VAR_GLOBAL
	// Interface ID for interface ITcVnCustomContainerOperation_ITcVnContainer
	{attribute 'tc_no_symbol'}
	IID_ITcVnCustomContainerOperation_ITcVnContainer: IID := (Data1 := 16#1324AA81, Data2 := 16#A16E, Data3 := 16#46B2, Data4 := [16#92, 16#D8, 16#11, 16#BE, 16#05, 16#66, 16#C7, 16#7A]);
	// Interface ID for interface ITcVnCustomContainerOperation_ITcVnForwardIterator
	{attribute 'tc_no_symbol'}
	IID_ITcVnCustomContainerOperation_ITcVnForwardIterator: IID := (Data1 := 16#C808A039, Data2 := 16#2D00, Data3 := 16#4B6B, Data4 := [16#89, 16#91, 16#24, 16#B1, 16#F3, 16#3D, 16#98, 16#7A]);
	// Interface ID for interface ITcVnCustomElementCondition_ITcVnContainer
	{attribute 'tc_no_symbol'}
	IID_ITcVnCustomElementCondition_ITcVnContainer: IID := (Data1 := 16#2529A58B, Data2 := 16#9E91, Data3 := 16#49A1, Data4 := [16#AD, 16#8A, 16#95, 16#06, 16#B8, 16#87, 16#F0, 16#65]);
	// Interface ID for interface ITcVnCustomElementCondition_ITcVnForwardIterator
	{attribute 'tc_no_symbol'}
	IID_ITcVnCustomElementCondition_ITcVnForwardIterator: IID := (Data1 := 16#7CF2DF09, Data2 := 16#9C9A, Data3 := 16#4433, Data4 := [16#98, 16#DD, 16#BF, 16#28, 16#40, 16#7D, 16#A3, 16#D4]);
	// Interface ID for interface ITcVnColorModel
	{attribute 'tc_no_symbol'}
	IID_ITcVnColorModel: IID := (Data1 := 16#0D1C5AC3, Data2 := 16#B759, Data3 := 16#4DFF, Data4 := [16#86, 16#24, 16#65, 16#78, 16#26, 16#E9, 16#F5, 16#8E]);
END_VAR

// Version/Global_Version
{attribute 'TcGenerated'}
// This function has been automatically generated from the project information.
VAR_GLOBAL CONSTANT
	{attribute 'const_non_replaced'}
	{attribute 'linkalways'}
	stLibVersion_Tc3_Vision : ST_LibVersion := (iMajor := 3, iMinor := 1, iBuild := 1, iRevision := 12, sVersion := '3.1.1.12');
	{attribute 'const_non_replaced'}
	{attribute 'linkalways'}
	sLibraryId_Tc3_Vision : String := 'Beckhoff Automation GmbH|Tc3_Vision|3.1.1.12';
END_VAR

// Global Variables/Global_Variables

	VAR_GLOBAL
		VISION_ADS_TIMEOUT	:	TIME := TIME#5s;	(* Default ADS timeout. *)
	END_VAR

// Function Blocks/Image Acquisition/FB_VN_GevCameraControl

	{attribute 'c++_compatible'}
	{attribute 'external_name' := 'FB_VN_GevCameraControl_GUID_F17A7C37_E616_4417_46AF_6CAA272D4BB4'}
	{attribute 'TcIecLibraryType'}
	(* This FB provides the basic functionality to control a GigE Vision camera and access its calibration data. *)
	FUNCTION_BLOCK FB_VN_GevCameraControl
	VAR
		(* Internal reference to the corresponding TcVnGevImageProvider TcCOM module ID, which needs to be set via TC init symbol. *)
		{attribute 'TcInitSymbol'}
		{attribute 'TcCategoryOID' := 'TcVnGevImageProvider'}
		 {attribute 'GUID' := '18071995-0000-0000-0000-00000000000F'}
		oidITcVnGevImageProvider : OTCID;
		 {attribute 'hide'}
		_reserved1 : UINT_0_32;
		(* Internal stuff *)
		{attribute 'hide'}
		 {attribute 'GUID' := '18071995-0000-0000-0000-000000000018'}
		pInternal : PVOID;
	END_VAR


	(* Delete all images contained in the TcVnGevImageProvider TcCOM module receive queue and reset the corresponding omitted images counter. *)
	METHOD ClearImageQueue : HRESULT
END_METHOD


	(* Close the control channel to the camera. *)
	METHOD CloseCamera : HRESULT
END_METHOD


	(* Internal method *)
	{attribute 'hide'}
	METHOD FB_exit : BOOL
	VAR_INPUT
		(*  if TRUE, the exit method is called for exiting an instance that is copied afterwards (online change). *)
		bInCopyCode : BOOL;
	END_VAR
END_METHOD


	(* Internal method *)
	{attribute 'hide'}
	METHOD FB_init : BOOL
	VAR_INPUT
		(*  if TRUE, the retain variables are initialized (warm start / cold start) *)
		bInitRetains : BOOL;
		(*  if TRUE, the instance afterwards gets moved into the copy code (online change) *)
		bInCopyCode : BOOL;
	END_VAR
END_METHOD


	(* Gets the reference calibration pattern points from the TcVnGevImageProvider TcCOM module (Can be set from the calibration assistant) *)
	METHOD GetCalibPatternRef : HRESULT
	VAR_INPUT
		(* Returns the reference calibration pattern points (ContainerType_Vector_TcVnPoint3_REAL) *)
 {attribute 'GUID' := 'BC72B333-E095-465B-9693-7979773CA3B8'}
				ipCalibPatternRef : REFERENCE TO ITcVnContainer;
	END_VAR
END_METHOD


	(* Gets the camera matrix from the TcVnGevImageProvider TcCOM module (requires intrinsic calibration parameters, e.g. set by the calibration assistant) *)
	METHOD GetCameraMatrix : HRESULT
	VAR_INPUT
		(* Returns the camera matrix *)
 {attribute 'GUID' := '91A420A3-4727-4481-B3BB-170528E5BC7C'}
		 {attribute 'Namespace' := 'VN'}
				aCameraMatrix : REFERENCE TO TcVnMatrix3x3_LREAL;
	END_VAR
END_METHOD


	(* Gets the current available image (first in receive queue). *)
	METHOD GetCurrentImage : HRESULT
	VAR_INPUT
		(* Returns the image *)
 {attribute 'GUID' := '70D42C6D-6F4E-4719-8B29-2883D5D59B1C'}
				ipImage : REFERENCE TO ITcVnImage;
	END_VAR
END_METHOD


	(* Gets the current available image (first in receive queue) with undistortion applied (requires intrinsic calibration parameters in the TcVnGevImageProvider TcCOM module, e.g. set by the calibration assistant) *)
	METHOD GetCurrentImageUndistorted : HRESULT
	VAR_INPUT
		(* Returns the undistorted image *)
 {attribute 'GUID' := '70D42C6D-6F4E-4719-8B29-2883D5D59B1C'}
				ipImage : REFERENCE TO ITcVnImage;
	END_VAR
END_METHOD


	(* Gets the current available image (first in receive queue) and its corresponding GVSP info. *)
	METHOD GetCurrentImageWithGvspInfo : HRESULT
	VAR_INPUT
		(* Returns the image *)
 {attribute 'GUID' := '70D42C6D-6F4E-4719-8B29-2883D5D59B1C'}
				ipImage : REFERENCE TO ITcVnImage;
		(* Returns the GVSP info *)
 {attribute 'GUID' := '63FC7E33-91CD-44CD-9015-0BD1DC25722C'}
				stGvspInfo : REFERENCE TO GVSP_IMAGE_INFO;
	END_VAR
END_METHOD


	(* Gets the current available image (first in receive queue) with its corresponding GVSP info and undistortion applied (requires intrinsic calibration parameters in the TcVnGevImageProvider TcCOM module, e.g. set by the calibration assistant) *)
	METHOD GetCurrentImageWithGvspInfoUndistorted : HRESULT
	VAR_INPUT
		(* Returns the undistorted image *)
 {attribute 'GUID' := '70D42C6D-6F4E-4719-8B29-2883D5D59B1C'}
				ipImage : REFERENCE TO ITcVnImage;
		(* Returns the GVSP info *)
 {attribute 'GUID' := '63FC7E33-91CD-44CD-9015-0BD1DC25722C'}
				stGvspInfo : REFERENCE TO GVSP_IMAGE_INFO;
	END_VAR
END_METHOD


	(* Gets the distortion coefficients from the TcVnGevImageProvider TcCOM module (requires intrinsic calibration parameters, e.g. set by the calibration assistant) *)
	METHOD GetDistortionCoefficients : HRESULT
	VAR_INPUT
		(* Returns the distortion coefficients [k1, k2, p1, p2, k3, k4, k5, k6] *)
 {attribute 'GUID' := 'DD112102-C23A-4B37-A43A-A96400B57010'}
		 {attribute 'Namespace' := 'VN'}
				aDistortionCoefficients : REFERENCE TO TcVnArray8_LREAL;
	END_VAR
END_METHOD


	(* Gets the last received image from the queue. *)
	METHOD GetLastImageFromQueue : HRESULT
	VAR_INPUT
		(* Returns the image *)
 {attribute 'GUID' := '70D42C6D-6F4E-4719-8B29-2883D5D59B1C'}
				ipImage : REFERENCE TO ITcVnImage;
	END_VAR
END_METHOD


	(* Gets the number of omitted images since the last call of ClearImageQueue(). If the image receive queue in the TcVnGevImageProvider TcCOM module is full and a new image arrives, the first one in the queue will be deleted and the omitted counter is increased. *)
	METHOD GetOmittedImagesNum : HRESULT
	VAR_INPUT
		(* Returns the number of omitted images *)
		nOmitted : REFERENCE TO ULINT;
	END_VAR
END_METHOD


	(* Gets the rotation matrix from the TcVnGevImageProvider TcCOM module (requires extrinsic calibration parameters, e.g. set by the calibration assistant) *)
	METHOD GetRotationMatrix : HRESULT
	VAR_INPUT
		(* Returns the rotation matrix *)
 {attribute 'GUID' := '91A420A3-4727-4481-B3BB-170528E5BC7C'}
		 {attribute 'Namespace' := 'VN'}
				aRotationMatrix : REFERENCE TO TcVnMatrix3x3_LREAL;
	END_VAR
END_METHOD


	(* Gets the current state of the internal camera control state machine. *)
	METHOD GetState : ETcVnCameraState
END_METHOD


	(* Gets the translation vector from the TcVnGevImageProvider TcCOM module (requires extrinsic calibration parameters, e.g. set by the calibration assistant) *)
	METHOD GetTranslationVector : HRESULT
	VAR_INPUT
		(* Returns the translation vector *)
 {attribute 'GUID' := 'B9A67DEB-A7D1-4F25-95A3-4A82FA5C1E28'}
		 {attribute 'Namespace' := 'VN'}
				aTranslationVector : REFERENCE TO TcVnVector3_LREAL;
	END_VAR
END_METHOD


	(* Initialize the camera to the intended state (includes sending the 'InitCameraCommands' defined in the GevImageAcquisition TcCOM module to the camera). *)
	METHOD InitializeCamera : HRESULT
END_METHOD


	(* Open a control channel to the camera. *)
	METHOD OpenCamera : HRESULT
END_METHOD


	(* Reset the camera controller to initial state (might require multiple calls depending on current state, until S_OK is returned) *)
	METHOD Reset : HRESULT
END_METHOD


	(* Reset the camera features to initial state (sends the 'InitCameraCommands' defined in the GevImageAcquisition TcCOM module to the camera). *)
	METHOD ResetCameraFeatures : HRESULT
END_METHOD


	(* Sets the camera matrix to the TcVnGevImageProvider TcCOM module *)
	METHOD SetCameraMatrix : HRESULT
	VAR_INPUT
		(* The camera matrix to be copied to the TcCOM module *)
 {attribute 'GUID' := '91A420A3-4727-4481-B3BB-170528E5BC7C'}
		 {attribute 'Namespace' := 'VN'}
				aCameraMatrix : REFERENCE TO TcVnMatrix3x3_LREAL;
	END_VAR
END_METHOD


	(* Sets the distortion coefficients to the TcVnGevImageProvider TcCOM module *)
	METHOD SetDistortionCoefficients : HRESULT
	VAR_INPUT
		(* The distortion coefficients to be copied to the TcCOM module *)
 {attribute 'GUID' := 'DD112102-C23A-4B37-A43A-A96400B57010'}
		 {attribute 'Namespace' := 'VN'}
				aDistortionCoefficients : REFERENCE TO TcVnArray8_LREAL;
	END_VAR
END_METHOD


	(* Sets the rotation matrix to the TcVnGevImageProvider TcCOM module *)
	METHOD SetRotationMatrix : HRESULT
	VAR_INPUT
		(* The rotation matrix to be copied to the TcCOM module *)
 {attribute 'GUID' := '91A420A3-4727-4481-B3BB-170528E5BC7C'}
		 {attribute 'Namespace' := 'VN'}
				aRotationMatrix : REFERENCE TO TcVnMatrix3x3_LREAL;
	END_VAR
END_METHOD


	(* Sets the translation vector to the TcVnGevImageProvider TcCOM module *)
	METHOD SetTranslationVector : HRESULT
	VAR_INPUT
		(* The translation vector to be copied to the TcCOM module *)
 {attribute 'GUID' := 'B9A67DEB-A7D1-4F25-95A3-4A82FA5C1E28'}
		 {attribute 'Namespace' := 'VN'}
				aTranslationVector : REFERENCE TO TcVnVector3_LREAL;
	END_VAR
END_METHOD


	(* Send the 'StartAcquisitionCommands' defined in the TcVnGevImageProvider TcCOM module to the camera. *)
	METHOD StartAcquisition : HRESULT
END_METHOD


	(* Send the 'StopAcquisitionCommands' defined in the TcVnGevImageProvider TcCOM module to the camera. *)
	METHOD StopAcquisition : HRESULT
END_METHOD


	(* Send the 'SoftwareTriggerCommands' defined in the TcVnGevImageProvider TcCOM module to the camera. *)
	METHOD TriggerImage : HRESULT
END_METHOD

END_FUNCTION_BLOCK

// Function Blocks/Image Acquisition/FB_VN_FileSourceControl

	{attribute 'c++_compatible'}
	{attribute 'external_name' := 'FB_VN_FileSourceControl_GUID_0F8A3DBC_2DD8_48DE_55D7_61CBFB8E01C0'}
	{attribute 'TcIecLibraryType'}
	(* This FB provides access to the images send by a File SOurce instance. *)
	FUNCTION_BLOCK FB_VN_FileSourceControl
	VAR
		(* Internal reference to the corresponding TcVnFileImageProvider TcCOM module ID, which needs to be set via TC init symbol. *)
		{attribute 'TcInitSymbol'}
		{attribute 'TcCategoryOID' := 'TcVnFileImageProvider'}
		 {attribute 'GUID' := '18071995-0000-0000-0000-00000000000F'}
		oidITcVnFileImageProvider : OTCID;
		 {attribute 'hide'}
		_reserved1 : UINT_0_32;
		(* Internal reference to private data. *)
		{attribute 'hide'}
		 {attribute 'GUID' := '18071995-0000-0000-0000-000000000018'}
		pPriv : PVOID;
	END_VAR


	(* Internal method *)
	{attribute 'hide'}
	METHOD FB_exit : BOOL
	VAR_INPUT
		(* If TRUE, the exit method is called for exiting an instance that is copied afterwards (online change). *)
		bInCopyCode : BOOL;
	END_VAR
END_METHOD


	(* Internal method *)
	{attribute 'hide'}
	METHOD FB_init : BOOL
	VAR_INPUT
		(* If TRUE, the retain variables are initialized (warm start / cold start) *)
		bInitRetains : BOOL;
		(* If TRUE, the exit method is called for exiting an instance that is copied afterwards (online change). *)
		bInCopyCode : BOOL;
	END_VAR
END_METHOD


	(* Gets the current available image (if any). *)
	METHOD GetCurrentImage : HRESULT
	VAR_INPUT
		(* Returns the image *)
 {attribute 'GUID' := '70D42C6D-6F4E-4719-8B29-2883D5D59B1C'}
				ipImage : REFERENCE TO ITcVnImage;
	END_VAR
END_METHOD


	(* Gets the current available image (if any) and the corresponding file name. *)
	METHOD GetCurrentImageAndFileName : HRESULT
	VAR_INPUT
		(* Returns the image *)
 {attribute 'GUID' := '70D42C6D-6F4E-4719-8B29-2883D5D59B1C'}
				ipImage : REFERENCE TO ITcVnImage;
	END_VAR
	VAR_IN_OUT CONSTANT
		(* Returns the file name *)
 {attribute 'GUID' := '18071995-0000-0000-0000-00000000001A'}
				sFileName : STRING;
	END_VAR
	VAR_INPUT
		(* Define the maximum allowed length for the file name *)
		nMaxLen : UINT;
	END_VAR
END_METHOD


	(* Activates the File Source. If not in trigger mode, it will start sending images. *)
	METHOD StartAcquisition : HRESULT
END_METHOD


	(* Deactivates the File Source. It will stop sending images. *)
	METHOD StopAcquisition : HRESULT
END_METHOD


	(* Reset the controller to initial state (might require multiple calls depending on current state, until S_OK is returned) *)
	METHOD Reset : HRESULT
END_METHOD


	(* Gets the current state of the internal camera control state machine. *)
	METHOD GetState : ETcVnCameraState
END_METHOD


	(* If in trigger mode, this function triggers the next image in the list. *)
	METHOD TriggerImage : HRESULT
END_METHOD


	(* If in trigger mode, this function triggers a specific image in the list. *)
	METHOD TriggerImageExp : HRESULT
	VAR_INPUT
		(* Amount of images to skip, relative to current *)
		nSkipImages : DINT;
	END_VAR
END_METHOD


	(* If in trigger mode, this function triggers a specific image in the list by name. *)
	METHOD TriggerImageByName : HRESULT
	VAR_IN_OUT CONSTANT
		(* Name of the image to trigger *)
 {attribute 'GUID' := '18071995-0000-0000-0000-00000000001A'}
				sImageName : STRING;
	END_VAR
END_METHOD

END_FUNCTION_BLOCK

// Function Blocks/Image Acquisition/FB_VN_SimpleCameraControl

	{attribute 'c++_compatible'}
	{attribute 'external_name' := 'FB_VN_SimpleCameraControl_GUID_85A4A3A7_7C55_424E_46D9_2337A2CE214C'}
	{attribute 'TcIecLibraryType'}
	(* This FB provides the basic functionality to control a camera or a FileSource. *)
	FUNCTION_BLOCK FB_VN_SimpleCameraControl
	VAR
		(* Internal reference to the corresponding TcVnImageProvider TcCOM module ID, which needs to be set via TC init symbol. *)
		{attribute 'TcInitSymbol'}
		{attribute 'TcCategoryOID' := 'TcVnImageProvider'}
		 {attribute 'GUID' := '18071995-0000-0000-0000-00000000000F'}
		oidITcVnImageProvider : OTCID;
		 {attribute 'hide'}
		_reserved1 : UINT_0_32;
		(* Internal stuff *)
		{attribute 'hide'}
		 {attribute 'GUID' := '18071995-0000-0000-0000-000000000018'}
		pInternal : PVOID;
	END_VAR


	(* Internal method *)
	{attribute 'hide'}
	METHOD FB_exit : BOOL
	VAR_INPUT
		(*  if TRUE, the exit method is called for exiting an instance that is copied afterwards (online change). *)
		bInCopyCode : BOOL;
	END_VAR
END_METHOD


	(* Internal method *)
	{attribute 'hide'}
	METHOD FB_init : BOOL
	VAR_INPUT
		(*  if TRUE, the retain variables are initialized (warm start / cold start) *)
		bInitRetains : BOOL;
		(*  if TRUE, the instance afterwards gets moved into the copy code (online change) *)
		bInCopyCode : BOOL;
	END_VAR
END_METHOD


	(* Get the current available image (if any). *)
	METHOD GetCurrentImage : HRESULT
	VAR_INPUT
		(* Returns the image *)
 {attribute 'GUID' := '70D42C6D-6F4E-4719-8B29-2883D5D59B1C'}
				ipImage : REFERENCE TO ITcVnImage;
	END_VAR
END_METHOD


	(* Get the current state of the internal camera control state machine. *)
	METHOD GetState : ETcVnCameraState
END_METHOD


	(* Reset the camera to initial state (might require multiple calls depending on current state, until S_OK is returned) *)
	METHOD Reset : HRESULT
END_METHOD


	(* Start the image acquisition. *)
	METHOD StartAcquisition : HRESULT
END_METHOD


	(* Stop the image acquisition. *)
	METHOD StopAcquisition : HRESULT
END_METHOD


	(* Trigger the next image. *)
	METHOD TriggerImage : HRESULT
END_METHOD

END_FUNCTION_BLOCK

// Function Blocks/File Access/FB_VN_ReadCalibrationPattern

	{attribute 'c++_compatible'}
	{attribute 'external_name' := 'FB_VN_ReadCalibrationPattern_GUID_B3A02584_AB5A_4ACE_53F2_D2DD5DC64051'}
	{attribute 'TcIecLibraryType'}
	(* This FB reads calibration pattern reference points from an xml file on the targte pc. *)
	FUNCTION_BLOCK FB_VN_ReadCalibrationPattern
	VAR_IN_OUT CONSTANT
		(* Full path of the file or relative path to the default directory on the target pc (%TWINCAT3DIR%\\CustomConfig\\Vision\\CalibrationPattern) *)
		 {attribute 'GUID' := '18071995-0000-0000-0000-00000000001A'}
		sFilePath : STRING;
	END_VAR
	VAR_INPUT
		(* Returns a container with the pattern points (ContainerType_Vector_TcVnPoint3_REAL) *)
		 {attribute 'GUID' := 'BC72B333-E095-465B-9693-7979773CA3B8'}
		ipDestContainer : REFERENCE TO ITcVnContainer;
		(* Reading the file is triggered by a rising edge at this input. *)
		bRead : BOOL;
	END_VAR
	VAR
		 {attribute 'hide'}
		_reserved1 : ARRAY [1..3] OF USINT;
	END_VAR
	VAR_INPUT
		(* Indicates the time before the function is cancelled. *)
		nTimeout : TIME := VISION_ADS_TIMEOUT;
	END_VAR
	VAR_OUTPUT
		(* This output remains TRUE until the function block has executed a command, but at the longest for the duration supplied to the 'nTimeout' input. While bBusy = TRUE, no new command will be accepted at the inputs. *)
		bBusy : BOOL;
		(* This output is switched to TRUE as soon as an error occurs during the execution of a command. The command-specific error code is contained in ‘nErrorId’. If the function block has a timeout error, 'bError' is TRUE and 'nErrorId' is 1861 (hexadecimal 0x745). Is reset to FALSE by the execution of a command at the inputs. *)
		bError : BOOL;
	END_VAR
	VAR
		 {attribute 'hide'}
		_reserved2 : UINT;
	END_VAR
	VAR_OUTPUT
		(* Contains the ADS error code or the command-specific error code of the last executed command. Is reset to 0 by the execution of a command at the inputs. *)
		nErrorId : UDINT;
	END_VAR
	VAR
		(* Internal parameter *)
		{attribute 'hide'}
		nAdsInvStamp : UINT;
		(* Internal parameter *)
		{attribute 'hide'}
		nAdsInvCnt : BYTE;
		(* Internal parameter *)
		{attribute 'hide'}
		ePendingRequest : BYTE;
		(* Internal parameter *)
		{attribute 'hide'}
		nTimeElapsed : TIME;
		(* Internal parameter *)
		{attribute 'hide'}
		bLastRead : BOOL;
		 {attribute 'hide'}
		_reserved3 : UINT_24_56;
		(* Internal parameter *)
		{attribute 'hide'}
		 {attribute 'GUID' := '18071995-0000-0000-0000-000000000018'}
		pBuffer : PVOID;
	END_VAR


	(* Internal method *)
	{attribute 'hide'}
	METHOD FB_exit : BOOL
	VAR_INPUT
		(*  if TRUE, the exit method is called for exiting an instance that is copied afterwards (online change). *)
		bInCopyCode : BOOL;
	END_VAR
END_METHOD


	(* Internal method *)
	{attribute 'hide'}
	METHOD FB_init : BOOL
	VAR_INPUT
		(*  if TRUE, the retain variables are initialized (warm start / cold start) *)
		bInitRetains : BOOL;
		(*  if TRUE, the instance afterwards gets moved into the copy code (online change) *)
		bInCopyCode : BOOL;
	END_VAR
END_METHOD

END_FUNCTION_BLOCK

// Function Blocks/File Access/FB_VN_ReadContainer

	{attribute 'c++_compatible'}
	{attribute 'external_name' := 'FB_VN_ReadContainer_GUID_4970374B_76DF_4A68_6AE7_EC922972F9F2'}
	{attribute 'TcIecLibraryType'}
	(* This FB reads a container from an xml file on the target pc. *)
	FUNCTION_BLOCK FB_VN_ReadContainer
	VAR_IN_OUT CONSTANT
		(* Full path of the file or relative path to the default directory on the target pc *)
		 {attribute 'GUID' := '18071995-0000-0000-0000-00000000001A'}
		sFilePath : STRING;
	END_VAR
	VAR_INPUT
		(* Returns a container with the loaded content *)
		 {attribute 'GUID' := 'BC72B333-E095-465B-9693-7979773CA3B8'}
		ipDestContainer : REFERENCE TO ITcVnContainer;
		(* The type id of the container to return. If this parameter is not set, a suitable container type will be determined automatically. *)
		 {attribute 'GUID' := '18071995-0000-0000-0000-000000000021'}
		nDestTypeGuid : GUID;
		(* Reading the file is triggered by a rising edge at this input. *)
		bRead : BOOL;
	END_VAR
	VAR
		 {attribute 'hide'}
		_reserved1 : ARRAY [1..3] OF USINT;
	END_VAR
	VAR_INPUT
		(* Indicates the time before the function is cancelled. *)
		nTimeout : TIME := VISION_ADS_TIMEOUT;
	END_VAR
	VAR_OUTPUT
		(* This output remains TRUE until the function block has executed a command, but at the longest for the duration supplied to the 'nTimeout' input. While bBusy = TRUE, no new command will be accepted at the inputs. *)
		bBusy : BOOL;
		(* This output is switched to TRUE as soon as an error occurs during the execution of a command. The command-specific error code is contained in ‘nErrorId’. If the function block has a timeout error, 'bError' is TRUE and 'nErrorId' is 1861 (hexadecimal 0x745). Is reset to FALSE by the execution of a command at the inputs. *)
		bError : BOOL;
	END_VAR
	VAR
		 {attribute 'hide'}
		_reserved2 : UINT;
	END_VAR
	VAR_OUTPUT
		(* Contains the ADS error code or the command-specific error code of the last executed command. Is reset to 0 by the execution of a command at the inputs. *)
		nErrorId : UDINT;
	END_VAR
	VAR
		(* Internal parameter *)
		{attribute 'hide'}
		nAdsInvStamp : UINT;
		(* Internal parameter *)
		{attribute 'hide'}
		nAdsInvCnt : BYTE;
		(* Internal parameter *)
		{attribute 'hide'}
		ePendingRequest : BYTE;
		(* Internal parameter *)
		{attribute 'hide'}
		nTimeElapsed : TIME;
		(* Internal parameter *)
		{attribute 'hide'}
		bLastRead : BOOL;
		 {attribute 'hide'}
		_reserved3 : UINT_24_56;
		(* Internal parameter *)
		{attribute 'hide'}
		 {attribute 'GUID' := '18071995-0000-0000-0000-000000000018'}
		pBuffer : PVOID;
	END_VAR


	(* Internal method *)
	{attribute 'hide'}
	METHOD FB_exit : BOOL
	VAR_INPUT
		(*  if TRUE, the exit method is called for exiting an instance that is copied afterwards (online change). *)
		bInCopyCode : BOOL;
	END_VAR
END_METHOD


	(* Internal method *)
	{attribute 'hide'}
	METHOD FB_init : BOOL
	VAR_INPUT
		(*  if TRUE, the retain variables are initialized (warm start / cold start) *)
		bInitRetains : BOOL;
		(*  if TRUE, the instance afterwards gets moved into the copy code (online change) *)
		bInCopyCode : BOOL;
	END_VAR
END_METHOD

END_FUNCTION_BLOCK

// Function Blocks/File Access/FB_VN_ReadImage

	{attribute 'c++_compatible'}
	{attribute 'external_name' := 'FB_VN_ReadImage_GUID_DC225DEA_0B37_4A85_7737_55D65C996AC9'}
	{attribute 'TcIecLibraryType'}
	(* This FB reads an image from a file on the target pc. *)
	FUNCTION_BLOCK FB_VN_ReadImage
	VAR_IN_OUT CONSTANT
		(* Full path of the file or relative path to the default image directory on the target pc *)
		 {attribute 'GUID' := '18071995-0000-0000-0000-00000000001A'}
		sFilePath : STRING;
	END_VAR
	VAR_INPUT
		(* Returns an image with the loaded content *)
		 {attribute 'GUID' := '70D42C6D-6F4E-4719-8B29-2883D5D59B1C'}
		ipDestImage : REFERENCE TO ITcVnImage;
		(* Reading the file is triggered by a rising edge at this input. *)
		bRead : BOOL;
	END_VAR
	VAR
		 {attribute 'hide'}
		_reserved1 : ARRAY [1..3] OF USINT;
	END_VAR
	VAR_INPUT
		(* Indicates the time before the function is cancelled. *)
		nTimeout : TIME := VISION_ADS_TIMEOUT;
	END_VAR
	VAR_OUTPUT
		(* This output remains TRUE until the function block has executed a command, but at the longest for the duration supplied to the 'nTimeout' input. While bBusy = TRUE, no new command will be accepted at the inputs. *)
		bBusy : BOOL;
		(* This output is switched to TRUE as soon as an error occurs during the execution of a command. The command-specific error code is contained in ‘nErrorId’. If the function block has a timeout error, 'bError' is TRUE and 'nErrorId' is 1861 (hexadecimal 0x745). Is reset to FALSE by the execution of a command at the inputs. *)
		bError : BOOL;
	END_VAR
	VAR
		 {attribute 'hide'}
		_reserved2 : UINT;
	END_VAR
	VAR_OUTPUT
		(* Contains the ADS error code or the command-specific error code of the last executed command. Is reset to 0 by the execution of a command at the inputs. *)
		nErrorId : UDINT;
	END_VAR
	VAR
		(* Internal parameter *)
		{attribute 'hide'}
		nAdsInvStamp : UINT;
		(* Internal parameter *)
		{attribute 'hide'}
		nAdsInvCnt : BYTE;
		(* Internal parameter *)
		{attribute 'hide'}
		ePendingRequest : BYTE;
		(* Internal parameter *)
		{attribute 'hide'}
		nTimeElapsed : TIME;
		(* Internal parameter *)
		{attribute 'hide'}
		bLastRead : BOOL;
		 {attribute 'hide'}
		_reserved3 : UINT_24_56;
		(* Internal parameter *)
		{attribute 'hide'}
		 {attribute 'GUID' := '18071995-0000-0000-0000-000000000018'}
		pBuffer : PVOID;
	END_VAR


	(* Internal method *)
	{attribute 'hide'}
	METHOD FB_exit : BOOL
	VAR_INPUT
		(*  if TRUE, the exit method is called for exiting an instance that is copied afterwards (online change). *)
		bInCopyCode : BOOL;
	END_VAR
END_METHOD


	(* Internal method *)
	{attribute 'hide'}
	METHOD FB_init : BOOL
	VAR_INPUT
		(*  if TRUE, the retain variables are initialized (warm start / cold start) *)
		bInitRetains : BOOL;
		(*  if TRUE, the instance afterwards gets moved into the copy code (online change) *)
		bInCopyCode : BOOL;
	END_VAR
END_METHOD

END_FUNCTION_BLOCK

// Function Blocks/File Access/FB_VN_WriteContainer

	{attribute 'c++_compatible'}
	{attribute 'external_name' := 'FB_VN_WriteContainer_GUID_7951D962_7694_4A6A_69EC_EB8831476B4E'}
	{attribute 'TcIecLibraryType'}
	(* This FB writes a container as an xml file to the hard drive. *)
	FUNCTION_BLOCK FB_VN_WriteContainer
	VAR_INPUT
		(* The container to write *)
		 {attribute 'GUID' := 'BC72B333-E095-465B-9693-7979773CA3B8'}
		ipContainer : ITcVnContainer;
	END_VAR
	VAR_IN_OUT CONSTANT
		(* Full path of the file or relative path to the default directory on the target pc *)
		 {attribute 'GUID' := '18071995-0000-0000-0000-00000000001A'}
		sFilePath : STRING;
	END_VAR
	VAR_INPUT
		(* Container export format (default is human readable xml) *)
		 {attribute 'GUID' := 'F8305D79-70A3-4F93-A939-2FF3B8D6AF74'}
		 {attribute 'Namespace' := 'Tc3_Vision'}
		eExportFormat : ETcVnContainerExportFormat := TCVN_CEF_XML;
		(* Writing the container is triggered by a rising edge at this input. *)
		bWrite : BOOL;
	END_VAR
	VAR
		 {attribute 'hide'}
		_reserved1 : USINT;
	END_VAR
	VAR_INPUT
		(* Indicates the time before the function is cancelled. *)
		nTimeout : TIME := VISION_ADS_TIMEOUT;
	END_VAR
	VAR_OUTPUT
		(* This output remains TRUE until the function block has executed a command, but at the longest for the duration supplied to the 'nTimeout' input. While bBusy = TRUE, no new command will be accepted at the inputs. *)
		bBusy : BOOL;
		(* This output is switched to TRUE as soon as an error occurs during the execution of a command. The command-specific error code is contained in ‘nErrorId’. If the function block has a timeout error, 'bError' is TRUE and 'nErrorId' is 1861 (hexadecimal 0x745). Is reset to FALSE by the execution of a command at the inputs. *)
		bError : BOOL;
	END_VAR
	VAR
		 {attribute 'hide'}
		_reserved2 : UINT;
	END_VAR
	VAR_OUTPUT
		(* Contains the ADS error code or the command-specific error code of the last executed command. Is reset to 0 by the execution of a command at the inputs. *)
		nErrorId : UDINT;
	END_VAR
	VAR
		(* Internal parameter *)
		{attribute 'hide'}
		nAdsInvStamp : UINT;
		(* Internal parameter *)
		{attribute 'hide'}
		nAdsInvCnt : BYTE;
		 {attribute 'hide'}
		_reserved3 : USINT;
		(* Internal parameter *)
		{attribute 'hide'}
		nTimeElapsed : TIME;
		(* Internal parameter *)
		{attribute 'hide'}
		bLastWrite : BOOL;
		 {attribute 'hide'}
		_reserved4 : UINT_24_56;
	END_VAR


	(* Internal method *)
	{attribute 'hide'}
	METHOD FB_exit : BOOL
	VAR_INPUT
		(* If TRUE, the exit method is called for exiting an instance that is copied afterwards (online change). *)
		bInCopyCode : BOOL;
	END_VAR
END_METHOD


	(* Internal method *)
	{attribute 'hide'}
	METHOD FB_init : BOOL
	VAR_INPUT
		(* If TRUE, the retain variables are initialized (warm start / cold start) *)
		bInitRetains : BOOL;
		(* If TRUE, the instance afterwards gets moved into the copy code (online change) *)
		bInCopyCode : BOOL;
	END_VAR
END_METHOD

END_FUNCTION_BLOCK

// Function Blocks/File Access/FB_VN_WriteImage

	{attribute 'c++_compatible'}
	{attribute 'external_name' := 'FB_VN_WriteImage_GUID_9751924C_ED9F_46AD_683F_5F581352D01B'}
	{attribute 'TcIecLibraryType'}
	(* This FB writes an image to the hard drive. *)
	FUNCTION_BLOCK FB_VN_WriteImage
	VAR_INPUT
		(* The image to write *)
		 {attribute 'GUID' := '70D42C6D-6F4E-4719-8B29-2883D5D59B1C'}
		ipImage : ITcVnImage;
	END_VAR
	VAR_IN_OUT CONSTANT
		(* If provided, the image is written to the given file path. Otherwise, if the string is empty, a default location specified by the connected service is used. *)
		 {attribute 'GUID' := '18071995-0000-0000-0000-00000000001A'}
		sFilePath : STRING;
	END_VAR
	VAR_INPUT
		(* Writing the image is triggered by a rising edge at this input. *)
		bWrite : BOOL;
	END_VAR
	VAR
		 {attribute 'hide'}
		_reserved1 : ARRAY [1..3] OF USINT;
	END_VAR
	VAR_INPUT
		(* Indicates the time before the function is cancelled. *)
		nTimeout : TIME := VISION_ADS_TIMEOUT;
	END_VAR
	VAR_OUTPUT
		(* This output remains TRUE until the function block has executed a command, but at the longest for the duration supplied to the 'nTimeout' input. While bBusy = TRUE, no new command will be accepted at the inputs. *)
		bBusy : BOOL;
		(* This output is switched to TRUE as soon as an error occurs during the execution of a command. The command-specific error code is contained in ‘nErrorId’. If the function block has a timeout error, 'bError' is TRUE and 'nErrorId' is 1861 (hexadecimal 0x745). Is reset to FALSE by the execution of a command at the inputs. *)
		bError : BOOL;
	END_VAR
	VAR
		 {attribute 'hide'}
		_reserved2 : UINT;
	END_VAR
	VAR_OUTPUT
		(* Contains the ADS error code or the command-specific error code of the last executed command. Is reset to 0 by the execution of a command at the inputs. *)
		nErrorId : UDINT;
	END_VAR
	VAR
		(* Internal parameter *)
		{attribute 'hide'}
		nAdsInvStamp : UINT;
		(* Internal parameter *)
		{attribute 'hide'}
		nAdsInvCnt : BYTE;
		 {attribute 'hide'}
		_reserved3 : USINT;
		(* Internal parameter *)
		{attribute 'hide'}
		nTimeElapsed : TIME;
		(* Internal parameter *)
		{attribute 'hide'}
		bLastWrite : BOOL;
		 {attribute 'hide'}
		_reserved4 : UINT_24_56;
	END_VAR


	(* Internal method *)
	{attribute 'hide'}
	METHOD FB_exit : BOOL
	VAR_INPUT
		(*  if TRUE, the exit method is called for exiting an instance that is copied afterwards (online change). *)
		bInCopyCode : BOOL;
	END_VAR
END_METHOD


	(* Internal method *)
	{attribute 'hide'}
	METHOD FB_init : BOOL
	VAR_INPUT
		(*  if TRUE, the retain variables are initialized (warm start / cold start) *)
		bInitRetains : BOOL;
		(*  if TRUE, the instance afterwards gets moved into the copy code (online change) *)
		bInCopyCode : BOOL;
	END_VAR
END_METHOD

END_FUNCTION_BLOCK

// Function Blocks/Camera Register Access/FB_VN_ReadRegister_UDINT

	{attribute 'c++_compatible'}
	{attribute 'external_name' := 'FB_VN_ReadRegister_UDINT_GUID_86A4A7D8_3848_4986_75BF_D4FFF92D82BE'}
	{attribute 'TcIecLibraryType'}
	(* This FB reads a DINT register from the camera. Requires an open control channel (e.g. by calling FB_VN_GevCameraControl.OpenCamera() before) *)
	FUNCTION_BLOCK FB_VN_ReadRegister_UDINT
	VAR_INPUT
		(* The address of the register that should be read *)
		 {attribute 'GUID' := 'E1ED2436-3512-43FA-B927-3F71DEDDA853'}
		nAddress : GVCP_REGISTER_ADDRESS;
		(* OPTIONAL: The endianness of the register. 0 = Big, 1 = Little. Default: 0 *)
		nEndian : UINT;
		(* Reading the register is triggered by a rising edge at this input. *)
		bRead : BOOL;
	END_VAR
	VAR
		 {attribute 'hide'}
		_reserved1 : USINT;
	END_VAR
	VAR_INPUT
		(* Indicates the time before the function is cancelled. *)
		nTimeout : TIME := VISION_ADS_TIMEOUT;
	END_VAR
	VAR_OUTPUT
		(* The read value *)
		nValue : UDINT;
		(* This output remains TRUE until the function block has executed a command, but at the longest for the duration supplied to the 'nTimeout' input. While bBusy = TRUE, no new command will be accepted at the inputs. *)
		bBusy : BOOL;
		(* This output is switched to TRUE as soon as an error occurs during the execution of a command. The command-specific error code is contained in ‘nErrorId’. If the function block has a timeout error, 'bError' is TRUE and 'nErrorId' is 1861 (hexadecimal 0x745). Is reset to FALSE by the execution of a command at the inputs. *)
		bError : BOOL;
	END_VAR
	VAR
		 {attribute 'hide'}
		_reserved2 : UINT;
	END_VAR
	VAR_OUTPUT
		(* Contains the ADS error code or the command-specific error code of the last executed command. Is reset to 0 by the execution of a command at the inputs. *)
		nErrorId : UDINT;
	END_VAR
	VAR
		{attribute 'TcInitSymbol'}
		{attribute 'TcCategoryOID' := 'TcVnGevImageProvider'}
		 {attribute 'GUID' := '18071995-0000-0000-0000-00000000000F'}
		oidITcVnGevImageProvider : OTCID;
		 {attribute 'hide'}
		_reserved3 : UINT_0_32;
		{attribute 'hide'}
		 {attribute 'GUID' := 'ED7659DB-95DC-4A4A-B62F-02C9870D5E81'}
		ipGevImageProvider : ITcVnGevImageProvider;
		{attribute 'hide'}
		nTimeElapsed : TIME;
		{attribute 'hide'}
		bLastRead : BOOL;
		 {attribute 'hide'}
		_reserved4 : ARRAY [1..3] OF USINT;
	END_VAR


	(* Internal method *)
	{attribute 'hide'}
	METHOD FB_exit : BOOL
	VAR_INPUT
		(*  if TRUE, the exit method is called for exiting an instance that is copied afterwards (online change). *)
		bInCopyCode : BOOL;
	END_VAR
END_METHOD


	(* Internal method *)
	{attribute 'hide'}
	METHOD FB_init : BOOL
	VAR_INPUT
		(*  if TRUE, the retain variables are initialized (warm start / cold start) *)
		bInitRetains : BOOL;
		(*  if TRUE, the instance afterwards gets moved into the copy code (online change) *)
		bInCopyCode : BOOL;
	END_VAR
END_METHOD

END_FUNCTION_BLOCK

// Function Blocks/Camera Register Access/FB_VN_WriteRegister_UDINT

	{attribute 'c++_compatible'}
	{attribute 'external_name' := 'FB_VN_WriteRegister_UDINT_GUID_98F89540_E30B_4324_6B7D_BA355BE96C1C'}
	{attribute 'TcIecLibraryType'}
	(* This FB writes a DINT value into a register on the camera. Requires an open control channel (e.g. by calling FB_VN_GevCameraControl.OpenCamera() before) *)
	FUNCTION_BLOCK FB_VN_WriteRegister_UDINT
	VAR_INPUT
		(* The address of the register that should be written *)
		 {attribute 'GUID' := 'E1ED2436-3512-43FA-B927-3F71DEDDA853'}
		nAddress : GVCP_REGISTER_ADDRESS;
		(* The value to write *)
		nValue : UDINT;
		(* OPTIONAL: The endianness of the register. 0 = Big, 1 = Little. Default: 0 *)
		nEndian : UINT;
		(* Reading the register is triggered by a rising edge at this input. *)
		bWrite : BOOL;
	END_VAR
	VAR
		 {attribute 'hide'}
		_reserved1 : USINT;
	END_VAR
	VAR_INPUT
		(* Indicates the time before the function is cancelled. *)
		nTimeout : TIME := VISION_ADS_TIMEOUT;
	END_VAR
	VAR_OUTPUT
		(* This output remains TRUE until the function block has executed a command, but at the longest for the duration supplied to the 'nTimeout' input. While bBusy = TRUE, no new command will be accepted at the inputs. *)
		bBusy : BOOL;
		(* This output is switched to TRUE as soon as an error occurs during the execution of a command. The command-specific error code is contained in ‘nErrorId’. If the function block has a timeout error, 'bError' is TRUE and 'nErrorId' is 1861 (hexadecimal 0x745). Is reset to FALSE by the execution of a command at the inputs. *)
		bError : BOOL;
	END_VAR
	VAR
		 {attribute 'hide'}
		_reserved2 : UINT;
	END_VAR
	VAR_OUTPUT
		(* Contains the ADS error code or the command-specific error code of the last executed command. Is reset to 0 by the execution of a command at the inputs. *)
		nErrorId : UDINT;
	END_VAR
	VAR
		{attribute 'TcInitSymbol'}
		{attribute 'TcCategoryOID' := 'TcVnGevImageProvider'}
		 {attribute 'GUID' := '18071995-0000-0000-0000-00000000000F'}
		oidITcVnGevImageProvider : OTCID;
		 {attribute 'hide'}
		_reserved3 : UINT_0_32;
		{attribute 'hide'}
		 {attribute 'GUID' := 'ED7659DB-95DC-4A4A-B62F-02C9870D5E81'}
		ipGevImageProvider : ITcVnGevImageProvider;
		{attribute 'hide'}
		nTimeElapsed : TIME;
		{attribute 'hide'}
		bLastWrite : BOOL;
		 {attribute 'hide'}
		_reserved4 : ARRAY [1..3] OF USINT;
	END_VAR


	(* Internal method *)
	{attribute 'hide'}
	METHOD FB_exit : BOOL
	VAR_INPUT
		(*  if TRUE, the exit method is called for exiting an instance that is copied afterwards (online change). *)
		bInCopyCode : BOOL;
	END_VAR
END_METHOD


	(* Internal method *)
	{attribute 'hide'}
	METHOD FB_init : BOOL
	VAR_INPUT
		(*  if TRUE, the retain variables are initialized (warm start / cold start) *)
		bInitRetains : BOOL;
		(*  if TRUE, the instance afterwards gets moved into the copy code (online change) *)
		bInCopyCode : BOOL;
	END_VAR
END_METHOD

END_FUNCTION_BLOCK

// Function Blocks/Camera Register Access/FB_VN_ReadMemory

	{attribute 'c++_compatible'}
	{attribute 'external_name' := 'FB_VN_ReadMemory_GUID_ABDD3EDA_D4E8_4525_4CAC_8287323CD5ED'}
	{attribute 'TcIecLibraryType'}
	(* This FB reads consecutive memory locations from the camera. Requires an open control channel (e.g. by calling FB_VN_GevCameraControl.OpenCamera() before) *)
	FUNCTION_BLOCK FB_VN_ReadMemory
	VAR_INPUT
		(* The address of the first byte to read from the camera (must be 32-bit aligned) *)
		 {attribute 'GUID' := 'E1ED2436-3512-43FA-B927-3F71DEDDA853'}
		nAddress : GVCP_REGISTER_ADDRESS;
		(* The number of bytes to read, starting with nAddress (must be a multiple of 4, not more than 536) *)
		nLength : UINT;
	END_VAR
	VAR
		 {attribute 'hide'}
		_reserved1 : UINT;
	END_VAR
	VAR_INPUT
		(* Pointer to the buffer where the read memory content is written to (The buffer must have a size of at least nLength bytes!) *)
		 {attribute 'GUID' := '18071995-0000-0000-0000-000000000018'}
		pBuffer : PVOID;
		(* Reading the memory is triggered by a rising edge at this input. *)
		bRead : BOOL;
	END_VAR
	VAR
		 {attribute 'hide'}
		_reserved2 : ARRAY [1..3] OF USINT;
	END_VAR
	VAR_INPUT
		(* Indicates the time before the function is cancelled. *)
		nTimeout : TIME := VISION_ADS_TIMEOUT;
	END_VAR
	VAR_OUTPUT
		(* This output remains TRUE until the function block has executed a command, but at the longest for the duration supplied to the 'nTimeout' input. While bBusy = TRUE, no new command will be accepted at the inputs. *)
		bBusy : BOOL;
		(* This output is switched to TRUE as soon as an error occurs during the execution of a command. The command-specific error code is contained in ‘nErrorId’. If the function block has a timeout error, 'bError' is TRUE and 'nErrorId' is 1861 (hexadecimal 0x745). Is reset to FALSE by the execution of a command at the inputs. *)
		bError : BOOL;
	END_VAR
	VAR
		 {attribute 'hide'}
		_reserved3 : UINT;
	END_VAR
	VAR_OUTPUT
		(* Contains the ADS error code or the command-specific error code of the last executed command. Is reset to 0 by the execution of a command at the inputs. *)
		nErrorId : UDINT;
	END_VAR
	VAR
		{attribute 'TcInitSymbol'}
		{attribute 'TcCategoryOID' := 'TcVnGevImageProvider'}
		 {attribute 'GUID' := '18071995-0000-0000-0000-00000000000F'}
		oidITcVnGevImageProvider : OTCID;
		 {attribute 'hide'}
		_reserved4 : UINT_0_32;
		{attribute 'hide'}
		 {attribute 'GUID' := 'ED7659DB-95DC-4A4A-B62F-02C9870D5E81'}
		ipGevImageProvider : ITcVnGevImageProvider;
		{attribute 'hide'}
		nTimeElapsed : TIME;
		{attribute 'hide'}
		bLastRead : BOOL;
		 {attribute 'hide'}
		_reserved5 : ARRAY [1..3] OF USINT;
	END_VAR


	(* Internal method *)
	{attribute 'hide'}
	METHOD FB_exit : BOOL
	VAR_INPUT
		(* If TRUE, the exit method is called for exiting an instance that is copied afterwards (online change). *)
		bInCopyCode : BOOL;
	END_VAR
END_METHOD


	(* Internal method *)
	{attribute 'hide'}
	METHOD FB_init : BOOL
	VAR_INPUT
		(* If TRUE, the retain variables are initialized (warm start / cold start) *)
		bInitRetains : BOOL;
		(* If TRUE, the instance afterwards gets moved into the copy code (online change) *)
		bInCopyCode : BOOL;
	END_VAR
END_METHOD

END_FUNCTION_BLOCK

// Function Blocks/Camera Register Access/FB_VN_WriteMemory

	{attribute 'c++_compatible'}
	{attribute 'external_name' := 'FB_VN_WriteMemory_GUID_BEFD2CC0_9DF1_4E01_5F27_4BBC7C7857B8'}
	{attribute 'TcIecLibraryType'}
	(* This FB writes data to consecutive memory locations on the camera. Requires an open control channel (e.g. by calling FB_VN_GevCameraControl.OpenCamera() before) *)
	FUNCTION_BLOCK FB_VN_WriteMemory
	VAR_INPUT
		(* The address of the first byte to write to the camera (must be 32-bit aligned) *)
		 {attribute 'GUID' := 'E1ED2436-3512-43FA-B927-3F71DEDDA853'}
		nAddress : GVCP_REGISTER_ADDRESS;
		(* The number of bytes to write, starting at nAddress (must be a multiple of 4, not more than 536) *)
		nLength : UINT;
	END_VAR
	VAR
		 {attribute 'hide'}
		_reserved1 : UINT;
	END_VAR
	VAR_INPUT
		(* Pointer to the data that should be written to the camera (must have a size of at least nLength bytes!) *)
		 {attribute 'GUID' := '18071995-0000-0000-0000-000000000018'}
		pData : PVOID;
		(* Writing the memory is triggered by a rising edge at this input. *)
		bWrite : BOOL;
	END_VAR
	VAR
		 {attribute 'hide'}
		_reserved2 : ARRAY [1..3] OF USINT;
	END_VAR
	VAR_INPUT
		(* Indicates the time before the function is cancelled. *)
		nTimeout : TIME := VISION_ADS_TIMEOUT;
	END_VAR
	VAR_OUTPUT
		(* This output remains TRUE until the function block has executed a command, but at the longest for the duration supplied to the 'nTimeout' input. While bBusy = TRUE, no new command will be accepted at the inputs. *)
		bBusy : BOOL;
		(* This output is switched to TRUE as soon as an error occurs during the execution of a command. The command-specific error code is contained in ‘nErrorId’. If the function block has a timeout error, 'bError' is TRUE and 'nErrorId' is 1861 (hexadecimal 0x745). Is reset to FALSE by the execution of a command at the inputs. *)
		bError : BOOL;
	END_VAR
	VAR
		 {attribute 'hide'}
		_reserved3 : UINT;
	END_VAR
	VAR_OUTPUT
		(* Contains the ADS error code or the command-specific error code of the last executed command. Is reset to 0 by the execution of a command at the inputs. *)
		nErrorId : UDINT;
		(* The number of bytes that have been successfully written to the camera. *)
		nBytesWritten : UINT;
	END_VAR
	VAR
		 {attribute 'hide'}
		_reserved4 : UINT;
		{attribute 'TcInitSymbol'}
		{attribute 'TcCategoryOID' := 'TcVnGevImageProvider'}
		 {attribute 'GUID' := '18071995-0000-0000-0000-00000000000F'}
		oidITcVnGevImageProvider : OTCID;
		{attribute 'hide'}
		 {attribute 'GUID' := 'ED7659DB-95DC-4A4A-B62F-02C9870D5E81'}
		ipGevImageProvider : ITcVnGevImageProvider;
		{attribute 'hide'}
		nTimeElapsed : TIME;
		{attribute 'hide'}
		bLastRead : BOOL;
		 {attribute 'hide'}
		_reserved5 : ARRAY [1..3] OF USINT;
	END_VAR


	(* Internal method *)
	{attribute 'hide'}
	METHOD FB_exit : BOOL
	VAR_INPUT
		(* If TRUE, the exit method is called for exiting an instance that is copied afterwards (online change). *)
		bInCopyCode : BOOL;
	END_VAR
END_METHOD


	(* Internal method *)
	{attribute 'hide'}
	METHOD FB_init : BOOL
	VAR_INPUT
		(* If TRUE, the retain variables are initialized (warm start / cold start) *)
		bInitRetains : BOOL;
		(* If TRUE, the instance afterwards gets moved into the copy code (online change) *)
		bInCopyCode : BOOL;
	END_VAR
END_METHOD

END_FUNCTION_BLOCK

// Function Blocks/Camera Register Access/FB_VN_ReadRegister_REAL

	{attribute 'c++_compatible'}
	{attribute 'external_name' := 'FB_VN_ReadRegister_REAL_GUID_DCE71FD4_537F_4A49_43F2_8ABE5BAAAD1D'}
	{attribute 'TcIecLibraryType'}
	(* This FB reads a REAL register from the camera. Requires an open control channel (e.g. by calling FB_VN_GevCameraControl.OpenCamera() before) *)
	FUNCTION_BLOCK FB_VN_ReadRegister_REAL
	VAR_INPUT
		(* The address of the register that should be read *)
		 {attribute 'GUID' := 'E1ED2436-3512-43FA-B927-3F71DEDDA853'}
		nAddress : GVCP_REGISTER_ADDRESS;
		(* OPTIONAL: The endianness of the register. 0 = Big, 1 = Little. Default: 0 *)
		nEndian : UINT;
		(* Reading the register is triggered by a rising edge at this input. *)
		bRead : BOOL;
	END_VAR
	VAR
		 {attribute 'hide'}
		_reserved1 : USINT;
	END_VAR
	VAR_INPUT
		(* Indicates the time before the function is cancelled. *)
		nTimeout : TIME := VISION_ADS_TIMEOUT;
	END_VAR
	VAR_OUTPUT
		(* The read value *)
		fValue : REAL;
		(* This output remains TRUE until the function block has executed a command, but at the longest for the duration supplied to the 'nTimeout' input. While bBusy = TRUE, no new command will be accepted at the inputs. *)
		bBusy : BOOL;
		(* This output is switched to TRUE as soon as an error occurs during the execution of a command. The command-specific error code is contained in ‘nErrorId’. If the function block has a timeout error, 'bError' is TRUE and 'nErrorId' is 1861 (hexadecimal 0x745). Is reset to FALSE by the execution of a command at the inputs. *)
		bError : BOOL;
	END_VAR
	VAR
		 {attribute 'hide'}
		_reserved2 : UINT;
	END_VAR
	VAR_OUTPUT
		(* Contains the ADS error code or the command-specific error code of the last executed command. Is reset to 0 by the execution of a command at the inputs. *)
		nErrorId : UDINT;
	END_VAR
	VAR
		{attribute 'TcInitSymbol'}
		{attribute 'TcCategoryOID' := 'TcVnGevImageProvider'}
		 {attribute 'GUID' := '18071995-0000-0000-0000-00000000000F'}
		oidITcVnGevImageProvider : OTCID;
		 {attribute 'hide'}
		_reserved3 : UINT_0_32;
		{attribute 'hide'}
		 {attribute 'GUID' := 'ED7659DB-95DC-4A4A-B62F-02C9870D5E81'}
		ipGevImageProvider : ITcVnGevImageProvider;
		{attribute 'hide'}
		nTimeElapsed : TIME;
		{attribute 'hide'}
		bLastRead : BOOL;
		 {attribute 'hide'}
		_reserved4 : ARRAY [1..3] OF USINT;
	END_VAR


	(* Internal method *)
	{attribute 'hide'}
	METHOD FB_exit : BOOL
	VAR_INPUT
		(*  if TRUE, the exit method is called for exiting an instance that is copied afterwards (online change). *)
		bInCopyCode : BOOL;
	END_VAR
END_METHOD


	(* Internal method *)
	{attribute 'hide'}
	METHOD FB_init : BOOL
	VAR_INPUT
		(*  if TRUE, the retain variables are initialized (warm start / cold start) *)
		bInitRetains : BOOL;
		(*  if TRUE, the instance afterwards gets moved into the copy code (online change) *)
		bInCopyCode : BOOL;
	END_VAR
END_METHOD

END_FUNCTION_BLOCK

// Function Blocks/Camera Register Access/FB_VN_WriteRegister_REAL

	{attribute 'c++_compatible'}
	{attribute 'external_name' := 'FB_VN_WriteRegister_REAL_GUID_CBE1CBAD_D403_433A_4619_9683135D5D08'}
	{attribute 'TcIecLibraryType'}
	(* This FB writes a REAL value into a register on the camera. Requires an open control channel (e.g. by calling FB_VN_GevCameraControl.OpenCamera() before) *)
	FUNCTION_BLOCK FB_VN_WriteRegister_REAL
	VAR_INPUT
		(* The address of the register that should be written *)
		 {attribute 'GUID' := 'E1ED2436-3512-43FA-B927-3F71DEDDA853'}
		nAddress : GVCP_REGISTER_ADDRESS;
		(* The value to write *)
		fValue : REAL;
		(* OPTIONAL: The endianness of the register. 0 = Big, 1 = Little. Default: 0 *)
		nEndian : UINT;
		(* Writing the register is triggered by a rising edge at this input. *)
		bWrite : BOOL;
	END_VAR
	VAR
		 {attribute 'hide'}
		_reserved1 : USINT;
	END_VAR
	VAR_INPUT
		(* Indicates the time before the function is cancelled. *)
		nTimeout : TIME := VISION_ADS_TIMEOUT;
	END_VAR
	VAR_OUTPUT
		(* This output remains TRUE until the function block has executed a command, but at the longest for the duration supplied to the 'nTimeout' input. While bBusy = TRUE, no new command will be accepted at the inputs. *)
		bBusy : BOOL;
		(* This output is switched to TRUE as soon as an error occurs during the execution of a command. The command-specific error code is contained in ‘nErrorId’. If the function block has a timeout error, 'bError' is TRUE and 'nErrorId' is 1861 (hexadecimal 0x745). Is reset to FALSE by the execution of a command at the inputs. *)
		bError : BOOL;
	END_VAR
	VAR
		 {attribute 'hide'}
		_reserved2 : UINT;
	END_VAR
	VAR_OUTPUT
		(* Contains the ADS error code or the command-specific error code of the last executed command. Is reset to 0 by the execution of a command at the inputs. *)
		nErrorId : UDINT;
	END_VAR
	VAR
		{attribute 'TcInitSymbol'}
		{attribute 'TcCategoryOID' := 'TcVnGevImageProvider'}
		 {attribute 'GUID' := '18071995-0000-0000-0000-00000000000F'}
		oidITcVnGevImageProvider : OTCID;
		 {attribute 'hide'}
		_reserved3 : UINT_0_32;
		{attribute 'hide'}
		 {attribute 'GUID' := 'ED7659DB-95DC-4A4A-B62F-02C9870D5E81'}
		ipGevImageProvider : ITcVnGevImageProvider;
		{attribute 'hide'}
		nTimeElapsed : TIME;
		{attribute 'hide'}
		bLastWrite : BOOL;
		 {attribute 'hide'}
		_reserved4 : ARRAY [1..3] OF USINT;
	END_VAR


	(* Internal method *)
	{attribute 'hide'}
	METHOD FB_exit : BOOL
	VAR_INPUT
		(*  if TRUE, the exit method is called for exiting an instance that is copied afterwards (online change). *)
		bInCopyCode : BOOL;
	END_VAR
END_METHOD


	(* Internal method *)
	{attribute 'hide'}
	METHOD FB_init : BOOL
	VAR_INPUT
		(*  if TRUE, the retain variables are initialized (warm start / cold start) *)
		bInitRetains : BOOL;
		(*  if TRUE, the instance afterwards gets moved into the copy code (online change) *)
		bInCopyCode : BOOL;
	END_VAR
END_METHOD

END_FUNCTION_BLOCK

// Functions/Control Functions/F_VN_StartAbsWatchdog

	{attribute 'TcIecLibraryType'}
	{attribute 'external_name' := 'F_VN_StartAbsWatchdog_GUID_6AA80BE6_658F_48D0_7621_CA4C8D60B5D6'}
	(* Starts a cooperative watchdog given an absolute stop time. *)
	FUNCTION F_VN_StartAbsWatchdog : HRESULT
	VAR_INPUT
		tStop	:	DINT;	(* Stop time in us *)
		hrPrev	:	HRESULT;	(* HRESULT indicating the result of previous operations (If SUCCEEDED(hrPrev) equals false, no operation is executed.) *)
	END_VAR

END_FUNCTION

// Functions/Control Functions/F_VN_StartAbsWatchdogExp

	{attribute 'TcIecLibraryType'}
	{attribute 'external_name' := 'F_VN_StartAbsWatchdogExp_GUID_FAE2FBB3_22C6_4444_5B94_541A9FD6D000'}
	(* Start a cooperative watchdog given an absolute stop time. (expert function) *)
	FUNCTION F_VN_StartAbsWatchdogExp : HRESULT
	VAR_INPUT
		tStop	:	DINT;	(* Stop time in us *)
		eWatchdogAccType	:	ETcWatchdogAccumulationType;	(* Accumalation method used for combining the results of multiple functions enclosed by this watchdog *)
		hrPrev	:	HRESULT;	(* HRESULT indicating the result of previous operations (If SUCCEEDED(hrPrev) equals false, no operation is executed.) *)
	END_VAR

END_FUNCTION

// Functions/Control Functions/F_VN_StartRelWatchdog

	{attribute 'TcIecLibraryType'}
	{attribute 'external_name' := 'F_VN_StartRelWatchdog_GUID_912B107F_57BF_4680_51B8_8A7E47D19E99'}
	(* Starts a cooperative watchdog given a stop time relative to the current time. *)
	FUNCTION F_VN_StartRelWatchdog : HRESULT
	VAR_INPUT
		tStop	:	DINT;	(* Stop time in us *)
		hrPrev	:	HRESULT;	(* HRESULT indicating the result of previous operations (If SUCCEEDED(hrPrev) equals false, no operation is executed.) *)
	END_VAR

END_FUNCTION

// Functions/Control Functions/F_VN_StartRelWatchdogExp

	{attribute 'TcIecLibraryType'}
	{attribute 'external_name' := 'F_VN_StartRelWatchdogExp_GUID_926BDD09_D519_4CB0_7417_0EF542A04680'}
	(* Start a cooperative watchdog given a stop time relative to the current time. (expert function) *)
	FUNCTION F_VN_StartRelWatchdogExp : HRESULT
	VAR_INPUT
		tStop	:	DINT;	(* Stop time in us *)
		eWatchdogAccType	:	ETcWatchdogAccumulationType;	(* Accumalation method used for combining the results of multiple functions enclosed by this watchdog *)
		hrPrev	:	HRESULT;	(* HRESULT indicating the result of previous operations (If SUCCEEDED(hrPrev) equals false, no operation is executed.) *)
	END_VAR

END_FUNCTION

// Functions/Control Functions/F_VN_StopWatchdog

	{attribute 'TcIecLibraryType'}
	{attribute 'external_name' := 'F_VN_StopWatchdog_GUID_F8F37EAF_3924_4731_4DFB_181063838513'}
	(* Stops a watchdog and provide runtime information. *)
	FUNCTION F_VN_StopWatchdog : HRESULT
	VAR_INPUT
		hrStartWatchdog	:	HRESULT;	(* HRESULT indicating the result of the function used to start the watchdog (If SUCCEEDED(hrStartWatchdog) equals false, no operation is executed.) *)
	END_VAR
	VAR_OUTPUT
		nFunctionsMonitored	:	ULINT;	(* Returns the number of functions monitored *)
		nFractionProcessed	:	UDINT;	(* Returns the fraction processed accumulated over the monitored functions in percent *)
		tRest	:	DINT;	(* Returns the remaining computation time in us (may be negative) *)
	END_VAR

END_FUNCTION

// Functions/Image Segmentation/F_VN_AdaptiveThreshold

	{attribute 'TcIecLibraryType'}
	{attribute 'external_name' := 'F_VN_AdaptiveThreshold_GUID_16A72604_B25C_4E1C_42EB_31A6D5D5EF8A'}
	(* Apply an adaptive threshold to a gray level image. *)
	FUNCTION F_VN_AdaptiveThreshold : HRESULT
	VAR_INPUT
		ipSrcImage	:	ITcVnImage;	(* Source image (1 channel, elements of type USINT) *)
		ipDestImage	:	REFERENCE TO ITcVnImage;	(* Destination image (An appropriate destination image will be created if required.) *)
		fMaxValue	:	LREAL;	(* Value assigned to pixels for which the threshold condition is true *)
		hrPrev	:	HRESULT;	(* HRESULT indicating the result of previous operations (If SUCCEEDED(hrPrev) equals false, no operation is executed.) *)
	END_VAR

END_FUNCTION

// Functions/Image Segmentation/F_VN_AdaptiveThresholdExp

	{attribute 'TcIecLibraryType'}
	{attribute 'external_name' := 'F_VN_AdaptiveThresholdExp_GUID_4305A328_4DB1_4A1A_45D9_927CE21EDCAE'}
	(* Apply an adaptive threshold to a gray level image. (expert function) *)
	FUNCTION F_VN_AdaptiveThresholdExp : HRESULT
	VAR_INPUT
		ipSrcImage	:	ITcVnImage;	(* Source image (1 channel, elements of type USINT) *)
		ipDestImage	:	REFERENCE TO ITcVnImage;	(* Destination image (An appropriate destination image will be created if required.) *)
		fMaxValue	:	LREAL;	(* Value assigned to pixels for which the threshold condition is true *)
		eAdaptiveMethod	:	ETcVnAdaptiveThresholdMethod;	(* Adaptive threshold method to be applied (MEAN: threshold value will be calculated as a mean of the nBlockSize x nBlockSize neighborhood of (x,y) minus fConstant. GAUSSIAN: threshold value is a weighted sum (cross-correlation with a Gaussian window) of the nBlockSize x nBlockSize neighborhood of (x,y) minus fConstant. *)
		eThresholdType	:	ETcVnThresholdType;	(* Threshold type to be applied (only BINARY and BINARY_INV are supported) *)
		nBlockSize	:	UDINT;	(* Size of the pixel neighborhood to calculate the local threshold (3, 5, 7, ...) *)
		fConstant	:	LREAL;	(* Constant that is subtracted from the weighted mean of the pixel neighborhood, which leads to the local threshold *)
		hrPrev	:	HRESULT;	(* HRESULT indicating the result of previous operations (If SUCCEEDED(hrPrev) equals false, no operation is executed.) *)
	END_VAR

END_FUNCTION

// Functions/Image Segmentation/F_VN_CheckColorRange

	{attribute 'TcIecLibraryType'}
	{attribute 'external_name' := 'F_VN_CheckColorRange_GUID_F81ECB61_09EB_44B1_51CE_375C171CBEC2'}
	(* Check if the pixel values of an image lie in a given range. The destination image has the same size as the source image but only one channel with
          a pixel element size of 8 bit. Its elements are set to 255 if the corresponding pixels of the source image are in the checked range and set to 0 otherwise. *)
	FUNCTION F_VN_CheckColorRange : HRESULT
	VAR_INPUT
		ipSrcImage	:	ITcVnImage;	(* Source image *)
		ipDestImage	:	REFERENCE TO ITcVnImage;	(* Destination image (An appropriate destination image will be created if required.) *)
		aLowerBounds	:	REFERENCE TO TcVnVector4_LREAL;	(* Channel-wise lower bounds (Unused channels are ignored.) *)
		aUpperBounds	:	REFERENCE TO TcVnVector4_LREAL;	(* Channel-wise upper bounds (Unused channels are ignored.) *)
		hrPrev	:	HRESULT;	(* HRESULT indicating the result of previous operations (If SUCCEEDED(hrPrev) equals false, no operation is executed.) *)
	END_VAR

END_FUNCTION

// Functions/Image Segmentation/F_VN_Threshold

	{attribute 'TcIecLibraryType'}
	{attribute 'external_name' := 'F_VN_Threshold_GUID_53A4D76B_53F9_45BC_75E9_9CF6A624606F'}
	(* Apply a fixed threshold or a dynamic threshold according to Otsu. *)
	FUNCTION F_VN_Threshold : HRESULT
	VAR_INPUT
		ipSrcImage	:	ITcVnImage;	(* Source image (1 channel) *)
		ipDestImage	:	REFERENCE TO ITcVnImage;	(* Destination image (An appropriate destination image will be created if required.) *)
		fThreshold	:	LREAL;	(* Fixed threshold (unused if dynamic thresholding is selected) *)
		fMaxValue	:	LREAL;	(* Maximum pixel value *)
		eThresholdType	:	ETcVnThresholdType;	(* Threshold type to be applied *)
		hrPrev	:	HRESULT;	(* HRESULT indicating the result of previous operations (If SUCCEEDED(hrPrev) equals false, no operation is executed.) *)
	END_VAR

END_FUNCTION

// Functions/Image Segmentation/F_VN_WatershedSegmentationExp

	{attribute 'TcIecLibraryType'}
	{attribute 'external_name' := 'F_VN_WatershedSegmentationExp_GUID_A25F1268_DD40_4E97_7B5F_71DED7FB685C'}
	(* Apply a marker-based watershed segmentation. (expert function) *)
	FUNCTION F_VN_WatershedSegmentationExp : HRESULT
	VAR_INPUT
		ipSrcImage	:	ITcVnImage;	(* Source image (USINT, 3 channels) *)
		ipDestImage	:	REFERENCE TO ITcVnImage;	(* Destination image (DINT, 1 channel. An appropriate image will be created if required.) *)
		ipMarkers	:	ITcVnImage;	(* Marker image (DINT, 1 channel) *)
		hrPrev	:	HRESULT;	(* HRESULT indicating the result of previous operations (If SUCCEEDED(hrPrev) equals false, no operation is executed.) *)
	END_VAR

END_FUNCTION

// Functions/Algebraic Image Operations/F_VN_AddImages

	{attribute 'TcIecLibraryType'}
	{attribute 'external_name' := 'F_VN_AddImages_GUID_C3D1AB7F_0DD2_484F_651B_09E60E401652'}
	(* Element-wise addition of two images using saturation arithmetics. *)
	FUNCTION F_VN_AddImages : HRESULT
	VAR_INPUT
		ipSrcImage1	:	ITcVnImage;	(* First source image *)
		ipSrcImage2	:	ITcVnImage;	(* Second source image *)
		ipDestImage	:	REFERENCE TO ITcVnImage;	(* Destination image (An appropriate destination image will be created if required.) *)
		hrPrev	:	HRESULT;	(* HRESULT indicating the result of previous operations (If SUCCEEDED(hrPrev) equals false, no operation is executed.) *)
	END_VAR

END_FUNCTION

// Functions/Algebraic Image Operations/F_VN_AddScalarToImage

	{attribute 'TcIecLibraryType'}
	{attribute 'external_name' := 'F_VN_AddScalarToImage_GUID_EF14740E_4720_4888_71A6_1EB9F42FEF7E'}
	(* Add a scalar value to each image pixel using saturation arithmetics. *)
	FUNCTION F_VN_AddScalarToImage : HRESULT
	VAR_INPUT
		fScalar	:	LREAL;	(* Scalar value *)
		ipSrcImage	:	ITcVnImage;	(* Source image *)
		ipDestImage	:	REFERENCE TO ITcVnImage;	(* Destination image (An appropriate destination image will be created if required.) *)
		hrPrev	:	HRESULT;	(* HRESULT indicating the result of previous operations (If SUCCEEDED(hrPrev) equals false, no operation is executed.) *)
	END_VAR

END_FUNCTION

// Functions/Algebraic Image Operations/F_VN_AddVectorToImage

	{attribute 'TcIecLibraryType'}
	{attribute 'external_name' := 'F_VN_AddVectorToImage_GUID_7A635C1A_8E29_4D4A_7267_E316E1F344FC'}
	(* Add a vector (1 element for each image channel) to each image pixel using saturation arithmetics. *)
	FUNCTION F_VN_AddVectorToImage : HRESULT
	VAR_INPUT
		aVector	:	REFERENCE TO TcVnVector4_LREAL;	(* 4-element vector (1 element for each image channel. If the image has less channels, the further vector elements are ignored.) *)
		ipSrcImage	:	ITcVnImage;	(* Source image *)
		ipDestImage	:	REFERENCE TO ITcVnImage;	(* Destination image (An appropriate destination image will be created if required.) *)
		hrPrev	:	HRESULT;	(* HRESULT indicating the result of previous operations (If SUCCEEDED(hrPrev) equals false, no operation is executed.) *)
	END_VAR

END_FUNCTION

// Functions/Algebraic Image Operations/F_VN_BitwiseAndImages

	{attribute 'TcIecLibraryType'}
	{attribute 'external_name' := 'F_VN_BitwiseAndImages_GUID_19C8EF47_5BE6_43F8_6E81_4653EE00BFBD'}
	(* Element-wise application of a bit-wise AND operator to two images. *)
	FUNCTION F_VN_BitwiseAndImages : HRESULT
	VAR_INPUT
		ipSrcImage1	:	ITcVnImage;	(* First source image *)
		ipSrcImage2	:	ITcVnImage;	(* Second source image *)
		ipDestImage	:	REFERENCE TO ITcVnImage;	(* Destination image (An appropriate destination image will be created if required.) *)
		hrPrev	:	HRESULT;	(* HRESULT indicating the result of previous operations (If SUCCEEDED(hrPrev) equals false, no operation is executed.) *)
	END_VAR

END_FUNCTION

// Functions/Algebraic Image Operations/F_VN_BitwiseAndImagesExp

	{attribute 'TcIecLibraryType'}
	{attribute 'external_name' := 'F_VN_BitwiseAndImagesExp_GUID_8F325577_61F2_40F0_5B4D_43869EB0485A'}
	(* Element-wise application of a bit-wise AND operator to two images. (expert function) *)
	FUNCTION F_VN_BitwiseAndImagesExp : HRESULT
	VAR_INPUT
		ipSrcImage1	:	ITcVnImage;	(* First source image *)
		ipSrcImage2	:	ITcVnImage;	(* Second source image *)
		ipDestImage	:	REFERENCE TO ITcVnImage;	(* Destination image (An appropriate destination image will be created if required.) *)
		ipMask	:	ITcVnImage;	(* Mask to limit the operation to specific pixel positions (mask value 0: skip pixel, mask value > 0: apply operation to pixel) *)
		hrPrev	:	HRESULT;	(* HRESULT indicating the result of previous operations (If SUCCEEDED(hrPrev) equals false, no operation is executed.) *)
	END_VAR

END_FUNCTION

// Functions/Algebraic Image Operations/F_VN_BitwiseAndScalarWithImage

	{attribute 'TcIecLibraryType'}
	{attribute 'external_name' := 'F_VN_BitwiseAndScalarWithImage_GUID_9F44F81B_708B_4CB6_7D2E_435C7DBE8615'}
	(* Bitwise and a scalar value with each image pixel. *)
	FUNCTION F_VN_BitwiseAndScalarWithImage : HRESULT
	VAR_INPUT
		fScalar	:	LREAL;	(* Scalar value *)
		ipSrcImage	:	ITcVnImage;	(* Source image *)
		ipDestImage	:	REFERENCE TO ITcVnImage;	(* Destination image (An appropriate destination image will be created if required.) *)
		hrPrev	:	HRESULT;	(* HRESULT indicating the result of previous operations (If SUCCEEDED(hrPrev) equals false, no operation is executed.) *)
	END_VAR

END_FUNCTION

// Functions/Algebraic Image Operations/F_VN_BitwiseAndVectorWithImage

	{attribute 'TcIecLibraryType'}
	{attribute 'external_name' := 'F_VN_BitwiseAndVectorWithImage_GUID_9B88B35E_CDB1_459D_42CA_0145D3EAAEEC'}
	(* Bitwise and a vector (1 element for each image channel) with each image pixel. *)
	FUNCTION F_VN_BitwiseAndVectorWithImage : HRESULT
	VAR_INPUT
		aVector	:	REFERENCE TO TcVnVector4_LREAL;	(* 4-element vector (1 element for each image channel. If the image has less channels, the further vector elements are ignored.) *)
		ipSrcImage	:	ITcVnImage;	(* Source image *)
		ipDestImage	:	REFERENCE TO ITcVnImage;	(* Destination image (An appropriate destination image will be created if required.) *)
		hrPrev	:	HRESULT;	(* HRESULT indicating the result of previous operations (If SUCCEEDED(hrPrev) equals false, no operation is executed.) *)
	END_VAR

END_FUNCTION

// Functions/Algebraic Image Operations/F_VN_BitwiseNotImage

	{attribute 'TcIecLibraryType'}
	{attribute 'external_name' := 'F_VN_BitwiseNotImage_GUID_A37ED9D0_F6EB_4E88_6B04_87BAAA365008'}
	(* Element-wise application of a bit-wise NOT operator to an image. *)
	FUNCTION F_VN_BitwiseNotImage : HRESULT
	VAR_INPUT
		ipSrcImage	:	ITcVnImage;	(* Source image *)
		ipDestImage	:	REFERENCE TO ITcVnImage;	(* Destination image (An appropriate destination image will be created if required.) *)
		hrPrev	:	HRESULT;	(* HRESULT indicating the result of previous operations (If SUCCEEDED(hrPrev) equals false, no operation is executed.) *)
	END_VAR

END_FUNCTION

// Functions/Algebraic Image Operations/F_VN_BitwiseNotImageExp

	{attribute 'TcIecLibraryType'}
	{attribute 'external_name' := 'F_VN_BitwiseNotImageExp_GUID_9D013208_88D7_411A_5E8B_1C99F5FBF99B'}
	(* Element-wise application of a bit-wise NOT operator to an image. (expert function) *)
	FUNCTION F_VN_BitwiseNotImageExp : HRESULT
	VAR_INPUT
		ipSrcImage	:	ITcVnImage;	(* Source image *)
		ipDestImage	:	REFERENCE TO ITcVnImage;	(* Destination image (An appropriate destination image will be created if required.) *)
		ipMask	:	ITcVnImage;	(* Mask to limit the operation to specific pixel positions (mask value 0: skip pixel, mask value > 0: apply operation to pixel) *)
		hrPrev	:	HRESULT;	(* HRESULT indicating the result of previous operations (If SUCCEEDED(hrPrev) equals false, no operation is executed.) *)
	END_VAR

END_FUNCTION

// Functions/Algebraic Image Operations/F_VN_BitwiseOrImages

	{attribute 'TcIecLibraryType'}
	{attribute 'external_name' := 'F_VN_BitwiseOrImages_GUID_6ED3E063_16FE_4CEC_4FBF_F95379A55CCC'}
	(* Element-wise application of a bit-wise OR operator to two images. *)
	FUNCTION F_VN_BitwiseOrImages : HRESULT
	VAR_INPUT
		ipSrcImage1	:	ITcVnImage;	(* First source image *)
		ipSrcImage2	:	ITcVnImage;	(* Second source image *)
		ipDestImage	:	REFERENCE TO ITcVnImage;	(* Destination image (An appropriate destination image will be created if required.) *)
		hrPrev	:	HRESULT;	(* HRESULT indicating the result of previous operations (If SUCCEEDED(hrPrev) equals false, no operation is executed.) *)
	END_VAR

END_FUNCTION

// Functions/Algebraic Image Operations/F_VN_BitwiseOrImagesExp

	{attribute 'TcIecLibraryType'}
	{attribute 'external_name' := 'F_VN_BitwiseOrImagesExp_GUID_C29D0E8C_900D_4055_4499_0EFC441D0CC1'}
	(* Element-wise application of a bit-wise OR operator to two images. (expert function) *)
	FUNCTION F_VN_BitwiseOrImagesExp : HRESULT
	VAR_INPUT
		ipSrcImage1	:	ITcVnImage;	(* First source image *)
		ipSrcImage2	:	ITcVnImage;	(* Second source image *)
		ipDestImage	:	REFERENCE TO ITcVnImage;	(* Destination image (An appropriate destination image will be created if required.) *)
		ipMask	:	ITcVnImage;	(* Mask to limit the operation to specific pixel positions (mask value 0: skip pixel, mask value > 0: apply operation to pixel) *)
		hrPrev	:	HRESULT;	(* HRESULT indicating the result of previous operations (If SUCCEEDED(hrPrev) equals false, no operation is executed.) *)
	END_VAR

END_FUNCTION

// Functions/Algebraic Image Operations/F_VN_BitwiseOrScalarWithImage

	{attribute 'TcIecLibraryType'}
	{attribute 'external_name' := 'F_VN_BitwiseOrScalarWithImage_GUID_A8566C54_991A_4FFB_58A5_4D525E068B46'}
	(* Bitwise or a scalar value with each image pixel. *)
	FUNCTION F_VN_BitwiseOrScalarWithImage : HRESULT
	VAR_INPUT
		fScalar	:	LREAL;	(* Scalar value *)
		ipSrcImage	:	ITcVnImage;	(* Source image *)
		ipDestImage	:	REFERENCE TO ITcVnImage;	(* Destination image (An appropriate destination image will be created if required.) *)
		hrPrev	:	HRESULT;	(* HRESULT indicating the result of previous operations (If SUCCEEDED(hrPrev) equals false, no operation is executed.) *)
	END_VAR

END_FUNCTION

// Functions/Algebraic Image Operations/F_VN_BitwiseOrVectorWithImage

	{attribute 'TcIecLibraryType'}
	{attribute 'external_name' := 'F_VN_BitwiseOrVectorWithImage_GUID_EF8EE95D_4380_42A7_7A5B_D1CBAE280EE3'}
	(* Bitwise or a vector (1 element for each image channel) with each image pixel. *)
	FUNCTION F_VN_BitwiseOrVectorWithImage : HRESULT
	VAR_INPUT
		aVector	:	REFERENCE TO TcVnVector4_LREAL;	(* 4-element vector (1 element for each image channel. If the image has less channels, the further vector elements are ignored.) *)
		ipSrcImage	:	ITcVnImage;	(* Source image *)
		ipDestImage	:	REFERENCE TO ITcVnImage;	(* Destination image (An appropriate destination image will be created if required.) *)
		hrPrev	:	HRESULT;	(* HRESULT indicating the result of previous operations (If SUCCEEDED(hrPrev) equals false, no operation is executed.) *)
	END_VAR

END_FUNCTION

// Functions/Algebraic Image Operations/F_VN_BitwiseXorImages

	{attribute 'TcIecLibraryType'}
	{attribute 'external_name' := 'F_VN_BitwiseXorImages_GUID_AF6BE629_E4FC_4C98_45BC_DD29A7F67719'}
	(* Element-wise application of a bit-wise XOR operator to two images. *)
	FUNCTION F_VN_BitwiseXorImages : HRESULT
	VAR_INPUT
		ipSrcImage1	:	ITcVnImage;	(* First source image *)
		ipSrcImage2	:	ITcVnImage;	(* Second source image *)
		ipDestImage	:	REFERENCE TO ITcVnImage;	(* Destination image (An appropriate destination image will be created if required.) *)
		hrPrev	:	HRESULT;	(* HRESULT indicating the result of previous operations (If SUCCEEDED(hrPrev) equals false, no operation is executed.) *)
	END_VAR

END_FUNCTION

// Functions/Algebraic Image Operations/F_VN_BitwiseXorImagesExp

	{attribute 'TcIecLibraryType'}
	{attribute 'external_name' := 'F_VN_BitwiseXorImagesExp_GUID_FC2A48D3_A5F5_4A8C_705F_B71CC93CC9C8'}
	(* Element-wise application of a bit-wise XOR operator to two images. (expert function) *)
	FUNCTION F_VN_BitwiseXorImagesExp : HRESULT
	VAR_INPUT
		ipSrcImage1	:	ITcVnImage;	(* First source image *)
		ipSrcImage2	:	ITcVnImage;	(* Second source image *)
		ipDestImage	:	REFERENCE TO ITcVnImage;	(* Destination image (An appropriate destination image will be created if required.) *)
		ipMask	:	ITcVnImage;	(* Mask to limit the operation to specific pixel positions (mask value 0: skip pixel, mask value > 0: apply operation to pixel) *)
		hrPrev	:	HRESULT;	(* HRESULT indicating the result of previous operations (If SUCCEEDED(hrPrev) equals false, no operation is executed.) *)
	END_VAR

END_FUNCTION

// Functions/Algebraic Image Operations/F_VN_BitwiseXorScalarWithImage

	{attribute 'TcIecLibraryType'}
	{attribute 'external_name' := 'F_VN_BitwiseXorScalarWithImage_GUID_96AFA1BD_7F68_4BEB_6255_7C6E88319FA7'}
	(* Bitwise xor a scalar value with each image pixel. *)
	FUNCTION F_VN_BitwiseXorScalarWithImage : HRESULT
	VAR_INPUT
		fScalar	:	LREAL;	(* Scalar value *)
		ipSrcImage	:	ITcVnImage;	(* Source image *)
		ipDestImage	:	REFERENCE TO ITcVnImage;	(* Destination image (An appropriate destination image will be created if required.) *)
		hrPrev	:	HRESULT;	(* HRESULT indicating the result of previous operations (If SUCCEEDED(hrPrev) equals false, no operation is executed.) *)
	END_VAR

END_FUNCTION

// Functions/Algebraic Image Operations/F_VN_BitwiseXorVectorWithImage

	{attribute 'TcIecLibraryType'}
	{attribute 'external_name' := 'F_VN_BitwiseXorVectorWithImage_GUID_10D91C57_F26F_4B77_661F_7AA13C332380'}
	(* Bitwise xor a vector (1 element for each image channel) with each image pixel. *)
	FUNCTION F_VN_BitwiseXorVectorWithImage : HRESULT
	VAR_INPUT
		aVector	:	REFERENCE TO TcVnVector4_LREAL;	(* 4-element vector (1 element for each image channel. If the image has less channels, the further vector elements are ignored.) *)
		ipSrcImage	:	ITcVnImage;	(* Source image *)
		ipDestImage	:	REFERENCE TO ITcVnImage;	(* Destination image (An appropriate destination image will be created if required.) *)
		hrPrev	:	HRESULT;	(* HRESULT indicating the result of previous operations (If SUCCEEDED(hrPrev) equals false, no operation is executed.) *)
	END_VAR

END_FUNCTION

// Functions/Algebraic Image Operations/F_VN_DivideImageByScalar

	{attribute 'TcIecLibraryType'}
	{attribute 'external_name' := 'F_VN_DivideImageByScalar_GUID_BF633759_801A_440D_515C_430C0CBCB74E'}
	(* Divide each image pixel by a scalar value using saturation arithmetics. *)
	FUNCTION F_VN_DivideImageByScalar : HRESULT
	VAR_INPUT
		ipSrcImage	:	ITcVnImage;	(* Source image *)
		fScalar	:	LREAL;	(* Scalar value *)
		ipDestImage	:	REFERENCE TO ITcVnImage;	(* Destination image (An appropriate destination image will be created if required.) *)
		hrPrev	:	HRESULT;	(* HRESULT indicating the result of previous operations (If SUCCEEDED(hrPrev) equals false, no operation is executed.) *)
	END_VAR

END_FUNCTION

// Functions/Algebraic Image Operations/F_VN_DivideImageByVector

	{attribute 'TcIecLibraryType'}
	{attribute 'external_name' := 'F_VN_DivideImageByVector_GUID_4F9CC9CA_F09C_49BB_5381_80C7E15F8806'}
	(* Divides each image pixel by a vector (1 element for each image channel) using saturation arithmetics. *)
	FUNCTION F_VN_DivideImageByVector : HRESULT
	VAR_INPUT
		ipSrcImage	:	ITcVnImage;	(* Source image *)
		aVector	:	REFERENCE TO TcVnVector4_LREAL;	(* 4-element vector (1 element for each image channel. If the image has less channels, the further vector elements are ignored.) *)
		ipDestImage	:	REFERENCE TO ITcVnImage;	(* Destination image (An appropriate destination image will be created if required.) *)
		hrPrev	:	HRESULT;	(* HRESULT indicating the result of previous operations (If SUCCEEDED(hrPrev) equals false, no operation is executed.) *)
	END_VAR

END_FUNCTION

// Functions/Algebraic Image Operations/F_VN_DivideImages

	{attribute 'TcIecLibraryType'}
	{attribute 'external_name' := 'F_VN_DivideImages_GUID_AF686B61_7ADF_4D38_5E5E_FA6F332C4D38'}
	(* Element-wise division of two images using saturation arithmetics. (A division by zero equals zero.) *)
	FUNCTION F_VN_DivideImages : HRESULT
	VAR_INPUT
		ipSrcImage1	:	ITcVnImage;	(* First source image (dividend) *)
		ipSrcImage2	:	ITcVnImage;	(* Second source image (divisor) *)
		ipDestImage	:	REFERENCE TO ITcVnImage;	(* Destination image (An appropriate destination image will be created if required.) *)
		hrPrev	:	HRESULT;	(* HRESULT indicating the result of previous operations (If SUCCEEDED(hrPrev) equals false, no operation is executed.) *)
	END_VAR

END_FUNCTION

// Functions/Algebraic Image Operations/F_VN_DivideScalarByImage

	{attribute 'TcIecLibraryType'}
	{attribute 'external_name' := 'F_VN_DivideScalarByImage_GUID_FC1D575C_B4CC_41E8_63F6_894807FE576F'}
	(* Divides a scalar value by each image pixel using saturation arithmetics. *)
	FUNCTION F_VN_DivideScalarByImage : HRESULT
	VAR_INPUT
		fScalar	:	LREAL;	(* Scalar value *)
		ipSrcImage	:	ITcVnImage;	(* Source image *)
		ipDestImage	:	REFERENCE TO ITcVnImage;	(* Destination image (An appropriate destination image will be created if required.) *)
		hrPrev	:	HRESULT;	(* HRESULT indicating the result of previous operations (If SUCCEEDED(hrPrev) equals false, no operation is executed.) *)
	END_VAR

END_FUNCTION

// Functions/Algebraic Image Operations/F_VN_DivideVectorByImage

	{attribute 'TcIecLibraryType'}
	{attribute 'external_name' := 'F_VN_DivideVectorByImage_GUID_F7383431_8202_45EE_53BB_CF59B8CE8AF7'}
	(* Divides a vector (1 element for each image channel) by each image pixel using saturation arithmetics. *)
	FUNCTION F_VN_DivideVectorByImage : HRESULT
	VAR_INPUT
		aVector	:	REFERENCE TO TcVnVector4_LREAL;	(* 4-element vector (1 element for each image channel. If the image has less channels, the further vector elements are ignored.) *)
		ipSrcImage	:	ITcVnImage;	(* Source image *)
		ipDestImage	:	REFERENCE TO ITcVnImage;	(* Destination image (An appropriate destination image will be created if required.) *)
		hrPrev	:	HRESULT;	(* HRESULT indicating the result of previous operations (If SUCCEEDED(hrPrev) equals false, no operation is executed.) *)
	END_VAR

END_FUNCTION

// Functions/Algebraic Image Operations/F_VN_ElementwiseExp

	{attribute 'TcIecLibraryType'}
	{attribute 'external_name' := 'F_VN_ElementwiseExp_GUID_D5D3EE2B_9CAD_453D_557A_248F03ABF7EE'}
	(* Computes the natural exponent of each pixel value. *)
	FUNCTION F_VN_ElementwiseExp : HRESULT
	VAR_INPUT
		ipSrcImage	:	ITcVnImage;	(* Source image *)
		ipDestImage	:	REFERENCE TO ITcVnImage;	(* Destination image (Same type and size as ipSrcImage, an appropriate image will be created if required.) *)
		hrPrev	:	HRESULT;	(* HRESULT indicating the result of previous operations (If SUCCEEDED(hrPrev) equals false, no operation is executed.) *)
	END_VAR

END_FUNCTION

// Functions/Algebraic Image Operations/F_VN_ElementwiseLog

	{attribute 'TcIecLibraryType'}
	{attribute 'external_name' := 'F_VN_ElementwiseLog_GUID_CD04F412_3E02_4323_6CCE_E9E57F40B5A7'}
	(* Computes the natural logarithm of each pixel value. *)
	FUNCTION F_VN_ElementwiseLog : HRESULT
	VAR_INPUT
		ipSrcImage	:	ITcVnImage;	(* Source image *)
		ipDestImage	:	REFERENCE TO ITcVnImage;	(* Destination image (Same type and size as ipSrcImage, an appropriate image will be created if required.) *)
		hrPrev	:	HRESULT;	(* HRESULT indicating the result of previous operations (If SUCCEEDED(hrPrev) equals false, no operation is executed.) *)
	END_VAR

END_FUNCTION

// Functions/Algebraic Image Operations/F_VN_MaxImage

	{attribute 'TcIecLibraryType'}
	{attribute 'external_name' := 'F_VN_MaxImage_GUID_AD4D7172_6019_47D7_6F67_EBCC8E97DBC2'}
	(* Element-wise maximum of two images. *)
	FUNCTION F_VN_MaxImage : HRESULT
	VAR_INPUT
		ipSrcImage1	:	ITcVnImage;	(* First source image *)
		ipSrcImage2	:	ITcVnImage;	(* Second source image *)
		ipDestImage	:	REFERENCE TO ITcVnImage;	(* Destination image (An appropriate destination image will be created if required.) *)
		hrPrev	:	HRESULT;	(* HRESULT indicating the result of previous operations (If SUCCEEDED(hrPrev) equals false, no operation is executed.) *)
	END_VAR

END_FUNCTION

// Functions/Algebraic Image Operations/F_VN_MaxImageExp

	{attribute 'TcIecLibraryType'}
	{attribute 'external_name' := 'F_VN_MaxImageExp_GUID_A300E46F_AA28_4C15_48A2_459D66C3EB1A'}
	(* Element-wise maximum of two images. (expert function) *)
	FUNCTION F_VN_MaxImageExp : HRESULT
	VAR_INPUT
		ipSrcImage1	:	ITcVnImage;	(* First source image *)
		ipSrcImage2	:	ITcVnImage;	(* Second source image *)
		ipDestImage	:	REFERENCE TO ITcVnImage;	(* Destination image (An appropriate destination image will be created if required.) *)
		ipMask	:	ITcVnImage;	(* Mask of type USINT *)
		hrPrev	:	HRESULT;	(* HRESULT indicating the result of previous operations (If SUCCEEDED(hrPrev) equals false, no operation is executed.) *)
	END_VAR

END_FUNCTION

// Functions/Algebraic Image Operations/F_VN_MaxImageWithScalar

	{attribute 'TcIecLibraryType'}
	{attribute 'external_name' := 'F_VN_MaxImageWithScalar_GUID_F88D0585_C233_4BA2_59E0_91626FE34716'}
	(* Element-wise maximum of image and scalar value. *)
	FUNCTION F_VN_MaxImageWithScalar : HRESULT
	VAR_INPUT
		fScalar	:	LREAL;	(* Scalar value *)
		ipSrcImage	:	ITcVnImage;	(* Source image *)
		ipDestImage	:	REFERENCE TO ITcVnImage;	(* Destination image (An appropriate destination image will be created if required.) *)
		hrPrev	:	HRESULT;	(* HRESULT indicating the result of previous operations (If SUCCEEDED(hrPrev) equals false, no operation is executed.) *)
	END_VAR

END_FUNCTION

// Functions/Algebraic Image Operations/F_VN_MaxImageWithScalarExp

	{attribute 'TcIecLibraryType'}
	{attribute 'external_name' := 'F_VN_MaxImageWithScalarExp_GUID_88BEAE48_2DB1_4562_5F88_1877D264AE84'}
	(* Element-wise maximum of image and scalar value. (expert function) *)
	FUNCTION F_VN_MaxImageWithScalarExp : HRESULT
	VAR_INPUT
		fScalar	:	LREAL;	(* Scalar value *)
		ipSrcImage	:	ITcVnImage;	(* Source image *)
		ipDestImage	:	REFERENCE TO ITcVnImage;	(* Destination image (An appropriate destination image will be created if required.) *)
		ipMask	:	ITcVnImage;	(* Mask of type USINT *)
		hrPrev	:	HRESULT;	(* HRESULT indicating the result of previous operations (If SUCCEEDED(hrPrev) equals false, no operation is executed.) *)
	END_VAR

END_FUNCTION

// Functions/Algebraic Image Operations/F_VN_MaxImageWithVector

	{attribute 'TcIecLibraryType'}
	{attribute 'external_name' := 'F_VN_MaxImageWithVector_GUID_1AFC8A8A_11EF_4CE0_4142_26B2D42C0D75'}
	(* Element-wise maximum of image and vector (1 element for each image channel). *)
	FUNCTION F_VN_MaxImageWithVector : HRESULT
	VAR_INPUT
		aVector	:	REFERENCE TO TcVnVector4_LREAL;	(* 4-element vector (1 element for each image channel. If the image has less channels, the further vector elements are ignored.) *)
		ipSrcImage	:	ITcVnImage;	(* Source image *)
		ipDestImage	:	REFERENCE TO ITcVnImage;	(* Destination image (An appropriate destination image will be created if required.) *)
		hrPrev	:	HRESULT;	(* HRESULT indicating the result of previous operations (If SUCCEEDED(hrPrev) equals false, no operation is executed.) *)
	END_VAR

END_FUNCTION

// Functions/Algebraic Image Operations/F_VN_MaxImageWithVectorExp

	{attribute 'TcIecLibraryType'}
	{attribute 'external_name' := 'F_VN_MaxImageWithVectorExp_GUID_0A11E948_8EAF_468A_4036_EA4CEFBA3ABA'}
	(* Element-wise maximum of image and vector (1 element for each image channel). (expert function) *)
	FUNCTION F_VN_MaxImageWithVectorExp : HRESULT
	VAR_INPUT
		aVector	:	REFERENCE TO TcVnVector4_LREAL;	(* 4-element vector (1 element for each image channel. If the image has less channels, the further vector elements are ignored.) *)
		ipSrcImage	:	ITcVnImage;	(* Source image *)
		ipDestImage	:	REFERENCE TO ITcVnImage;	(* Destination image (An appropriate destination image will be created if required.) *)
		ipMask	:	ITcVnImage;	(* Mask of type USINT *)
		hrPrev	:	HRESULT;	(* HRESULT indicating the result of previous operations (If SUCCEEDED(hrPrev) equals false, no operation is executed.) *)
	END_VAR

END_FUNCTION

// Functions/Algebraic Image Operations/F_VN_MinImage

	{attribute 'TcIecLibraryType'}
	{attribute 'external_name' := 'F_VN_MinImage_GUID_CDD55A16_3DC2_4993_4426_CA742076F425'}
	(* Element-wise minimum of two images. *)
	FUNCTION F_VN_MinImage : HRESULT
	VAR_INPUT
		ipSrcImage1	:	ITcVnImage;	(* First source image *)
		ipSrcImage2	:	ITcVnImage;	(* Second source image *)
		ipDestImage	:	REFERENCE TO ITcVnImage;	(* Destination image (An appropriate destination image will be created if required.) *)
		hrPrev	:	HRESULT;	(* HRESULT indicating the result of previous operations (If SUCCEEDED(hrPrev) equals false, no operation is executed.) *)
	END_VAR

END_FUNCTION

// Functions/Algebraic Image Operations/F_VN_MinImageExp

	{attribute 'TcIecLibraryType'}
	{attribute 'external_name' := 'F_VN_MinImageExp_GUID_29148138_4312_4CCF_716F_B410E7C9228D'}
	(* Element-wise minimum of two images. (expert function) *)
	FUNCTION F_VN_MinImageExp : HRESULT
	VAR_INPUT
		ipSrcImage1	:	ITcVnImage;	(* First source image *)
		ipSrcImage2	:	ITcVnImage;	(* Second source image *)
		ipDestImage	:	REFERENCE TO ITcVnImage;	(* Destination image (An appropriate destination image will be created if required.) *)
		ipMask	:	ITcVnImage;	(* Mask of type USINT *)
		hrPrev	:	HRESULT;	(* HRESULT indicating the result of previous operations (If SUCCEEDED(hrPrev) equals false, no operation is executed.) *)
	END_VAR

END_FUNCTION

// Functions/Algebraic Image Operations/F_VN_MinImageWithScalar

	{attribute 'TcIecLibraryType'}
	{attribute 'external_name' := 'F_VN_MinImageWithScalar_GUID_200C4856_8FCD_4F8E_6CCD_D1CD452EFB30'}
	(* Element-wise minimum of image and scalar value. *)
	FUNCTION F_VN_MinImageWithScalar : HRESULT
	VAR_INPUT
		fScalar	:	LREAL;	(* Scalar value *)
		ipSrcImage	:	ITcVnImage;	(* Source image *)
		ipDestImage	:	REFERENCE TO ITcVnImage;	(* Destination image (An appropriate destination image will be created if required.) *)
		hrPrev	:	HRESULT;	(* HRESULT indicating the result of previous operations (If SUCCEEDED(hrPrev) equals false, no operation is executed.) *)
	END_VAR

END_FUNCTION

// Functions/Algebraic Image Operations/F_VN_MinImageWithScalarExp

	{attribute 'TcIecLibraryType'}
	{attribute 'external_name' := 'F_VN_MinImageWithScalarExp_GUID_E51B4F15_0750_43A2_6D67_56E9240A9075'}
	(* Element-wise minimum of image and scalar value. (expert function) *)
	FUNCTION F_VN_MinImageWithScalarExp : HRESULT
	VAR_INPUT
		fScalar	:	LREAL;	(* Scalar value *)
		ipSrcImage	:	ITcVnImage;	(* Source image *)
		ipDestImage	:	REFERENCE TO ITcVnImage;	(* Destination image (An appropriate destination image will be created if required.) *)
		ipMask	:	ITcVnImage;	(* Mask of type USINT *)
		hrPrev	:	HRESULT;	(* HRESULT indicating the result of previous operations (If SUCCEEDED(hrPrev) equals false, no operation is executed.) *)
	END_VAR

END_FUNCTION

// Functions/Algebraic Image Operations/F_VN_MinImageWithVector

	{attribute 'TcIecLibraryType'}
	{attribute 'external_name' := 'F_VN_MinImageWithVector_GUID_01C10B47_9C6B_4A3B_7A92_2A3BCA1E20EA'}
	(* Element-wise minimum of image and vector (1 element for each image channel). *)
	FUNCTION F_VN_MinImageWithVector : HRESULT
	VAR_INPUT
		aVector	:	REFERENCE TO TcVnVector4_LREAL;	(* 4-element vector (1 element for each image channel. If the image has less channels, the further vector elements are ignored.) *)
		ipSrcImage	:	ITcVnImage;	(* Source image *)
		ipDestImage	:	REFERENCE TO ITcVnImage;	(* Destination image (An appropriate destination image will be created if required.) *)
		hrPrev	:	HRESULT;	(* HRESULT indicating the result of previous operations (If SUCCEEDED(hrPrev) equals false, no operation is executed.) *)
	END_VAR

END_FUNCTION

// Functions/Algebraic Image Operations/F_VN_MinImageWithVectorExp

	{attribute 'TcIecLibraryType'}
	{attribute 'external_name' := 'F_VN_MinImageWithVectorExp_GUID_AEAE8CCE_1BBB_4641_4EC9_AD3C80242FFF'}
	(* Element-wise minimum of image and vector (1 element for each image channel). (expert function) *)
	FUNCTION F_VN_MinImageWithVectorExp : HRESULT
	VAR_INPUT
		aVector	:	REFERENCE TO TcVnVector4_LREAL;	(* 4-element vector (1 element for each image channel. If the image has less channels, the further vector elements are ignored.) *)
		ipSrcImage	:	ITcVnImage;	(* Source image *)
		ipDestImage	:	REFERENCE TO ITcVnImage;	(* Destination image (An appropriate destination image will be created if required.) *)
		ipMask	:	ITcVnImage;	(* Mask of type USINT *)
		hrPrev	:	HRESULT;	(* HRESULT indicating the result of previous operations (If SUCCEEDED(hrPrev) equals false, no operation is executed.) *)
	END_VAR

END_FUNCTION

// Functions/Algebraic Image Operations/F_VN_MultiplyImages

	{attribute 'TcIecLibraryType'}
	{attribute 'external_name' := 'F_VN_MultiplyImages_GUID_5E667F0F_DF1B_47EC_431B_D728AB6B230A'}
	(* Element-wise multiplication of two images using saturation arithmetics. *)
	FUNCTION F_VN_MultiplyImages : HRESULT
	VAR_INPUT
		ipSrcImage1	:	ITcVnImage;	(* First source image *)
		ipSrcImage2	:	ITcVnImage;	(* Second source image *)
		ipDestImage	:	REFERENCE TO ITcVnImage;	(* Destination image (An appropriate destination image will be created if required.) *)
		hrPrev	:	HRESULT;	(* HRESULT indicating the result of previous operations (If SUCCEEDED(hrPrev) equals false, no operation is executed.) *)
	END_VAR

END_FUNCTION

// Functions/Algebraic Image Operations/F_VN_MultiplyImageWithScalar

	{attribute 'TcIecLibraryType'}
	{attribute 'external_name' := 'F_VN_MultiplyImageWithScalar_GUID_6DE705BC_07BA_4B8A_5F9D_F0F19A04EA0B'}
	(* Multiply each image pixel by a scalar value using saturation arithmetics. *)
	FUNCTION F_VN_MultiplyImageWithScalar : HRESULT
	VAR_INPUT
		fScalar	:	LREAL;	(* Scalar value *)
		ipSrcImage	:	ITcVnImage;	(* Source image *)
		ipDestImage	:	REFERENCE TO ITcVnImage;	(* Destination image (An appropriate destination image will be created if required.) *)
		hrPrev	:	HRESULT;	(* HRESULT indicating the result of previous operations (If SUCCEEDED(hrPrev) equals false, no operation is executed.) *)
	END_VAR

END_FUNCTION

// Functions/Algebraic Image Operations/F_VN_MultiplyImageWithVector

	{attribute 'TcIecLibraryType'}
	{attribute 'external_name' := 'F_VN_MultiplyImageWithVector_GUID_869A8BBA_69EC_4CD8_68E8_712F457C2053'}
	(* Multiply each image pixel by a vector (1 element for each image channel) using saturation arithmetics. *)
	FUNCTION F_VN_MultiplyImageWithVector : HRESULT
	VAR_INPUT
		aVector	:	REFERENCE TO TcVnVector4_LREAL;	(* 4-element vector (1 element for each image channel. If the image has less channels, the further vector elements are ignored.) *)
		ipSrcImage	:	ITcVnImage;	(* Source image *)
		ipDestImage	:	REFERENCE TO ITcVnImage;	(* Destination image (An appropriate destination image will be created if required.) *)
		hrPrev	:	HRESULT;	(* HRESULT indicating the result of previous operations (If SUCCEEDED(hrPrev) equals false, no operation is executed.) *)
	END_VAR

END_FUNCTION

// Functions/Algebraic Image Operations/F_VN_SubtractImageFromScalar

	{attribute 'TcIecLibraryType'}
	{attribute 'external_name' := 'F_VN_SubtractImageFromScalar_GUID_64660544_71D5_4932_6CDB_D0FCB0F60670'}
	(* Subtract each image pixel from a scalar value using saturation arithmetics. *)
	FUNCTION F_VN_SubtractImageFromScalar : HRESULT
	VAR_INPUT
		fScalar	:	LREAL;	(* Scalar value *)
		ipSrcImage	:	ITcVnImage;	(* Source image *)
		ipDestImage	:	REFERENCE TO ITcVnImage;	(* Destination image (An appropriate destination image will be created if required.) *)
		hrPrev	:	HRESULT;	(* HRESULT indicating the result of previous operations (If SUCCEEDED(hrPrev) equals false, no operation is executed.) *)
	END_VAR

END_FUNCTION

// Functions/Algebraic Image Operations/F_VN_SubtractImageFromVector

	{attribute 'TcIecLibraryType'}
	{attribute 'external_name' := 'F_VN_SubtractImageFromVector_GUID_CB9D587B_9393_45CD_7DAF_07D041E353B5'}
	(* Subtract each image pixel from a vector (1 element for each image channel) using saturation arithmetics. *)
	FUNCTION F_VN_SubtractImageFromVector : HRESULT
	VAR_INPUT
		aVector	:	REFERENCE TO TcVnVector4_LREAL;	(* 4-element vector (1 element for each image channel. If the image has less channels, the further vector elements are ignored.) *)
		ipSrcImage	:	ITcVnImage;	(* Source image *)
		ipDestImage	:	REFERENCE TO ITcVnImage;	(* Destination image (An appropriate destination image will be created if required.) *)
		hrPrev	:	HRESULT;	(* HRESULT indicating the result of previous operations (If SUCCEEDED(hrPrev) equals false, no operation is executed.) *)
	END_VAR

END_FUNCTION

// Functions/Algebraic Image Operations/F_VN_SubtractImages

	{attribute 'TcIecLibraryType'}
	{attribute 'external_name' := 'F_VN_SubtractImages_GUID_4F670E94_6A2E_4150_6F75_97E5E6BF17A6'}
	(* Element-wise subtraction of two images using saturation arithmetics. *)
	FUNCTION F_VN_SubtractImages : HRESULT
	VAR_INPUT
		ipSrcImage1	:	ITcVnImage;	(* First source image (minuend) *)
		ipSrcImage2	:	ITcVnImage;	(* Second source image (subtrahend) *)
		ipDestImage	:	REFERENCE TO ITcVnImage;	(* Destination image (An appropriate destination image will be created if required.) *)
		hrPrev	:	HRESULT;	(* HRESULT indicating the result of previous operations (If SUCCEEDED(hrPrev) equals false, no operation is executed.) *)
	END_VAR

END_FUNCTION

// Functions/Algebraic Image Operations/F_VN_SubtractScalarFromImage

	{attribute 'TcIecLibraryType'}
	{attribute 'external_name' := 'F_VN_SubtractScalarFromImage_GUID_96B9E213_5CA9_481C_7034_03FAC2495952'}
	(* Subtract a scalar value from each image pixel using saturation arithmetics. *)
	FUNCTION F_VN_SubtractScalarFromImage : HRESULT
	VAR_INPUT
		ipSrcImage	:	ITcVnImage;	(* Source image *)
		fScalar	:	LREAL;	(* Scalar value *)
		ipDestImage	:	REFERENCE TO ITcVnImage;	(* Destination image (An appropriate destination image will be created if required.) *)
		hrPrev	:	HRESULT;	(* HRESULT indicating the result of previous operations (If SUCCEEDED(hrPrev) equals false, no operation is executed.) *)
	END_VAR

END_FUNCTION

// Functions/Algebraic Image Operations/F_VN_SubtractVectorFromImage

	{attribute 'TcIecLibraryType'}
	{attribute 'external_name' := 'F_VN_SubtractVectorFromImage_GUID_E6892A3F_E280_4B9B_7676_40D6549E6D29'}
	(* Subtract a vector (1 element for each image channel) from each image pixel using saturation arithmetics. *)
	FUNCTION F_VN_SubtractVectorFromImage : HRESULT
	VAR_INPUT
		ipSrcImage	:	ITcVnImage;	(* Source image *)
		aVector	:	REFERENCE TO TcVnVector4_LREAL;	(* 4-element vector (1 element for each image channel. If the image has less channels, the further vector elements are ignored.) *)
		ipDestImage	:	REFERENCE TO ITcVnImage;	(* Destination image (An appropriate destination image will be created if required.) *)
		hrPrev	:	HRESULT;	(* HRESULT indicating the result of previous operations (If SUCCEEDED(hrPrev) equals false, no operation is executed.) *)
	END_VAR

END_FUNCTION

// Functions/Image Analysis/F_VN_CannyEdgeDetection

	{attribute 'TcIecLibraryType'}
	{attribute 'external_name' := 'F_VN_CannyEdgeDetection_GUID_719D53D7_E08D_4EB8_7439_78A761FEB067'}
	(* Find edges using the Canny edge detection algorithm. *)
	FUNCTION F_VN_CannyEdgeDetection : HRESULT
	VAR_INPUT
		ipSrcImage	:	ITcVnImage;	(* Source image (elements of type USINT) *)
		ipDestImage	:	REFERENCE TO ITcVnImage;	(* Destination image (elements of type USINT. An appropriate destination image will be created if required.) *)
		fThresholdLow	:	LREAL;	(* Low threshold *)
		fThresholdHigh	:	LREAL;	(* High threshold *)
		hrPrev	:	HRESULT;	(* HRESULT indicating the result of previous operations (If SUCCEEDED(hrPrev) equals false, no operation is executed.) *)
	END_VAR

END_FUNCTION

// Functions/Image Analysis/F_VN_CannyEdgeDetectionExp

	{attribute 'TcIecLibraryType'}
	{attribute 'external_name' := 'F_VN_CannyEdgeDetectionExp_GUID_B1C486F5_1123_4BDE_4220_A347DFC73D09'}
	(* Find edges using the Canny edge detection algorithm. (expert function) *)
	FUNCTION F_VN_CannyEdgeDetectionExp : HRESULT
	VAR_INPUT
		ipSrcImage	:	ITcVnImage;	(* Source image (elements of type USINT) *)
		ipDestImage	:	REFERENCE TO ITcVnImage;	(* Destination image (elements of type USINT. An appropriate destination image will be created if required.) *)
		fThresholdLow	:	LREAL;	(* Low threshold *)
		fThresholdHigh	:	LREAL;	(* High threshold *)
		nApertureSize	:	UDINT;	(* Aperture size for the Sobel operator (3, 5, 7) *)
		bL2Gradient	:	BOOL;	(* If true, the more accurate (and slower) L2 norm is used instead of the L1 norm *)
		hrPrev	:	HRESULT;	(* HRESULT indicating the result of previous operations (If SUCCEEDED(hrPrev) equals false, no operation is executed.) *)
	END_VAR

END_FUNCTION

// Functions/Image Analysis/F_VN_CountNonZeroPixels

	{attribute 'TcIecLibraryType'}
	{attribute 'external_name' := 'F_VN_CountNonZeroPixels_GUID_41EBF67E_B621_4A59_78FD_E05EDF933898'}
	(* Counts the non-zero pixels in a single-channel image (e.g. useful to analyze threshold results). *)
	FUNCTION F_VN_CountNonZeroPixels : HRESULT
	VAR_INPUT
		ipSrcImage	:	ITcVnImage;	(* Source image (1 channel) *)
		nNonZero	:	REFERENCE TO ULINT;	(* Returns the number of non-zero pixels in ipSrcImage *)
		hrPrev	:	HRESULT;	(* HRESULT indicating the result of previous operations (If SUCCEEDED(hrPrev) equals false, no operation is executed.) *)
	END_VAR

END_FUNCTION

// Functions/Image Analysis/F_VN_DistanceTransformation

	{attribute 'TcIecLibraryType'}
	{attribute 'external_name' := 'F_VN_DistanceTransformation_GUID_9256B5BA_2753_4BE3_4382_59676EE6EE03'}
	(* Calculates the distance transformation, which is the distance to the closest zero pixel in a binary image. *)
	FUNCTION F_VN_DistanceTransformation : HRESULT
	VAR_INPUT
		ipSrcImage	:	ITcVnImage;	(* Source image (USINT, 1 channel) *)
		ipDestImage	:	REFERENCE TO ITcVnImage;	(* Destination image (REAL, 1 channel. An appropriate destination image will be created if required.) *)
		eDistanceType	:	ETcVnDistanceType;	(* Distance computation method (supported: L1, L2, C) *)
		eMaskSize	:	ETcVnDistanceTransformationMask;	(* Size of the distance transformation mask *)
		hrPrev	:	HRESULT;	(* HRESULT indicating the result of previous operations (If SUCCEEDED(hrPrev) equals false, no operation is executed.) *)
	END_VAR

END_FUNCTION

// Functions/Image Analysis/F_VN_DistanceTransformationExp

	{attribute 'TcIecLibraryType'}
	{attribute 'external_name' := 'F_VN_DistanceTransformationExp_GUID_90311457_1B37_4ACC_720F_989CF5A12C11'}
	(* Calculates the distance transformation, which is the distance to the closest zero pixel in a binary image. Additionally, an image with component labels is created (discrete Voronoi diagram). (expert function) *)
	FUNCTION F_VN_DistanceTransformationExp : HRESULT
	VAR_INPUT
		ipSrcImage	:	ITcVnImage;	(* Source image (USINT, 1 channel) *)
		ipDestImage	:	REFERENCE TO ITcVnImage;	(* Destination image (REAL, 1 channel. An appropriate destination image will be created if required.) *)
		eDistanceType	:	ETcVnDistanceType;	(* Distance computation method (supported: L1, L2, C) *)
		eMaskSize	:	ETcVnDistanceTransformationMask;	(* Size of the distance transformation mask (PRECISE not supported for label computation) *)
		ipDestLabels	:	REFERENCE TO ITcVnImage;	(* Returns the component labels (Discrete Voronoi diagram; DINT, 1 channel. An appropriate image will be created if required.) *)
		eLabelType	:	ETcVnDistanceTransformationLabel;	(* Type of the labels *)
		hrPrev	:	HRESULT;	(* HRESULT indicating the result of previous operations (If SUCCEEDED(hrPrev) equals false, no operation is executed.) *)
	END_VAR

END_FUNCTION

// Functions/Image Analysis/F_VN_ImageAverage

	{attribute 'TcIecLibraryType'}
	{attribute 'external_name' := 'F_VN_ImageAverage_GUID_D10E9A22_CE1F_4851_43C2_0BECED86D006'}
	(* Computes the (channel-wise) average pixel value of an image. *)
	FUNCTION F_VN_ImageAverage : HRESULT
	VAR_INPUT
		ipSrcImage	:	ITcVnImage;	(* Source image (1 - 4 channels) *)
		aAverage	:	REFERENCE TO TcVnVector4_LREAL;	(* Returns the (channel-wise) average pixel value of ipSrcImage *)
		hrPrev	:	HRESULT;	(* HRESULT indicating the result of previous operations (If SUCCEEDED(hrPrev) equals false, no operation is executed.) *)
	END_VAR

END_FUNCTION

// Functions/Image Analysis/F_VN_ImageAverageExp

	{attribute 'TcIecLibraryType'}
	{attribute 'external_name' := 'F_VN_ImageAverageExp_GUID_11587096_3748_40F4_624D_16522BA4497D'}
	(* Computes the (channel-wise) average pixel value of an image. (expert function) *)
	FUNCTION F_VN_ImageAverageExp : HRESULT
	VAR_INPUT
		ipSrcImage	:	ITcVnImage;	(* Source image (1 - 4 channels) *)
		aAverage	:	REFERENCE TO TcVnVector4_LREAL;	(* Returns the (channel-wise) average pixel value of ipSrcImage *)
		ipMask	:	ITcVnImage;	(* Mask of type USINT (1 channel) *)
		hrPrev	:	HRESULT;	(* HRESULT indicating the result of previous operations (If SUCCEEDED(hrPrev) equals false, no operation is executed.) *)
	END_VAR

END_FUNCTION

// Functions/Image Analysis/F_VN_ImageAverageStdDev

	{attribute 'TcIecLibraryType'}
	{attribute 'external_name' := 'F_VN_ImageAverageStdDev_GUID_E6CA9AFB_86EA_4EBD_461C_7F6A20F0B932'}
	(* Computes the (channel-wise) average pixel value and the corresponding standard deviation of an image. *)
	FUNCTION F_VN_ImageAverageStdDev : HRESULT
	VAR_INPUT
		ipSrcImage	:	ITcVnImage;	(* Source image (1 - 4 channels) *)
		aAverage	:	REFERENCE TO TcVnVector4_LREAL;	(* Returns the (channel-wise) average pixel value of ipSrcImage *)
		aStdDev	:	REFERENCE TO TcVnVector4_LREAL;	(* Returns the (channel-wise) pixel value standard deviation of ipSrcImage *)
		hrPrev	:	HRESULT;	(* HRESULT indicating the result of previous operations (If SUCCEEDED(hrPrev) equals false, no operation is executed.) *)
	END_VAR

END_FUNCTION

// Functions/Image Analysis/F_VN_ImageAverageStdDevExp

